(* Logix 5000 project; controller reports 1756-L63 rev 20.11; software revision 20.04; part 7 of 52 *)

        [627].log_data[17].valid := 1, [627].log_data[18].valid := 1, [627].log_data[19].valid := 1, [627].time.Year := 2023, [627].time.Month := 1, [627].time.Day := 14, [627].time.Hour := 5, [627].time.Minute := 14, [627].time.Second := 59, [628].log_data[0].min := 1.0, [628].log_data[0].max := 1.0, [628].log_data[0].total := 900.0, [628].log_data[0].time := 900.0, [628].log_data[0].minminute := 15, [628].log_data[0].maxminute := 15, [628].log_data[0].valid := 1, [628].log_data[1].valid := 1, [628].log_data[2].valid := 1, [628].log_data[3].valid := 1, [628].log_data[4].valid := 1, [628].log_data[5].valid := 1, [628].log_data[6].valid := 1, [628].log_data[7].valid := 1, [628].log_data[8].valid := 1, [628].log_data[9].valid := 1, [628].log_data[10].valid := 1, [628].log_data[11].valid := 1, [628].log_data[12].valid := 1, [628].log_data[13].valid := 1, [628].log_data[14].valid := 1, [628].log_data[15].valid := 1, [628].log_data[16].valid := 1, [628].log_data[17].valid := 1, [628].log_data[18].valid := 1, [628].log_data[19].valid := 1, [628].time.Year := 2023, [628].time.Month := 1, [628].time.Day := 14, [628].time.Hour := 5, [628].time.Minute := 29, [628].time.Second := 59, [629].log_data[0].min := 1.0, [629].log_data[0].max := 1.0, [629].log_data[0].total := 900.0, [629].log_data[0].time := 900.0, [629].log_data[0].minminute := 30, [629].log_data[0].maxminute := 30, [629].log_data[0].valid := 1, [629].log_data[1].valid := 1, [629].log_data[2].valid := 1, [629].log_data[3].valid := 1, [629].log_data[4].valid := 1, [629].log_data[5].valid := 1, [629].log_data[6].valid := 1, [629].log_data[7].valid := 1, [629].log_data[8].valid := 1, [629].log_data[9].valid := 1, [629].log_data[10].valid := 1, [629].log_data[11].valid := 1, [629].log_data[12].valid := 1,
        [629].log_data[13].valid := 1, [629].log_data[14].valid := 1, [629].log_data[15].valid := 1, [629].log_data[16].valid := 1, [629].log_data[17].valid := 1, [629].log_data[18].valid := 1, [629].log_data[19].valid := 1, [629].time.Year := 2023, [629].time.Month := 1, [629].time.Day := 14, [629].time.Hour := 5, [629].time.Minute := 44, [629].time.Second := 59, [630].log_data[0].min := 1.0, [630].log_data[0].max := 1.0, [630].log_data[0].total := 900.0, [630].log_data[0].time := 900.0, [630].log_data[0].minminute := 45, [630].log_data[0].maxminute := 45, [630].log_data[0].valid := 1, [630].log_data[1].valid := 1, [630].log_data[2].valid := 1, [630].log_data[3].valid := 1, [630].log_data[4].valid := 1, [630].log_data[5].valid := 1, [630].log_data[6].valid := 1, [630].log_data[7].valid := 1, [630].log_data[8].valid := 1, [630].log_data[9].valid := 1, [630].log_data[10].valid := 1, [630].log_data[11].valid := 1, [630].log_data[12].valid := 1, [630].log_data[13].valid := 1, [630].log_data[14].valid := 1, [630].log_data[15].valid := 1, [630].log_data[16].valid := 1, [630].log_data[17].valid := 1, [630].log_data[18].valid := 1, [630].log_data[19].valid := 1, [630].time.Year := 2023, [630].time.Month := 1, [630].time.Day := 14, [630].time.Hour := 5, [630].time.Minute := 59, [630].time.Second := 59, [631].log_data[0].min := 1.0, [631].log_data[0].max := 1.0, [631].log_data[0].total := 900.0, [631].log_data[0].time := 900.0, [631].log_data[0].valid := 1, [631].log_data[1].valid := 1, [631].log_data[2].valid := 1, [631].log_data[3].valid := 1, [631].log_data[4].valid := 1, [631].log_data[5].valid := 1, [631].log_data[6].valid := 1, [631].log_data[7].valid := 1, [631].log_data[8].valid := 1, [631].log_data[9].valid := 1, [631].log_data[10].valid := 1,
        [631].log_data[11].valid := 1, [631].log_data[12].valid := 1, [631].log_data[13].valid := 1, [631].log_data[14].valid := 1, [631].log_data[15].valid := 1, [631].log_data[16].valid := 1, [631].log_data[17].valid := 1, [631].log_data[18].valid := 1, [631].log_data[19].valid := 1, [631].time.Year := 2023, [631].time.Month := 1, [631].time.Day := 14, [631].time.Hour := 6, [631].time.Minute := 14, [631].time.Second := 59, [632].log_data[0].min := 1.0, [632].log_data[0].max := 1.0, [632].log_data[0].total := 900.0, [632].log_data[0].time := 900.0, [632].log_data[0].minminute := 15, [632].log_data[0].maxminute := 15, [632].log_data[0].valid := 1, [632].log_data[1].valid := 1, [632].log_data[2].valid := 1, [632].log_data[3].valid := 1, [632].log_data[4].valid := 1, [632].log_data[5].valid := 1, [632].log_data[6].valid := 1, [632].log_data[7].valid := 1, [632].log_data[8].valid := 1, [632].log_data[9].valid := 1, [632].log_data[10].valid := 1, [632].log_data[11].valid := 1, [632].log_data[12].valid := 1, [632].log_data[13].valid := 1, [632].log_data[14].valid := 1, [632].log_data[15].valid := 1, [632].log_data[16].valid := 1, [632].log_data[17].valid := 1, [632].log_data[18].valid := 1, [632].log_data[19].valid := 1, [632].time.Year := 2023, [632].time.Month := 1, [632].time.Day := 14, [632].time.Hour := 6, [632].time.Minute := 29, [632].time.Second := 59, [633].log_data[0].min := 1.0, [633].log_data[0].max := 1.0, [633].log_data[0].total := 900.0, [633].log_data[0].time := 900.0, [633].log_data[0].minminute := 30, [633].log_data[0].maxminute := 30, [633].log_data[0].valid := 1, [633].log_data[1].valid := 1, [633].log_data[2].valid := 1, [633].log_data[3].valid := 1, [633].log_data[4].valid := 1, [633].log_data[5].valid := 1, [633].log_data[6].valid := 1,
        [633].log_data[7].valid := 1, [633].log_data[8].valid := 1, [633].log_data[9].valid := 1, [633].log_data[10].valid := 1, [633].log_data[11].valid := 1, [633].log_data[12].valid := 1, [633].log_data[13].valid := 1, [633].log_data[14].valid := 1, [633].log_data[15].valid := 1, [633].log_data[16].valid := 1, [633].log_data[17].valid := 1, [633].log_data[18].valid := 1, [633].log_data[19].valid := 1, [633].time.Year := 2023, [633].time.Month := 1, [633].time.Day := 14, [633].time.Hour := 6, [633].time.Minute := 44, [633].time.Second := 59, [634].log_data[0].min := 1.0, [634].log_data[0].max := 1.0, [634].log_data[0].total := 900.0, [634].log_data[0].time := 900.0, [634].log_data[0].minminute := 45, [634].log_data[0].maxminute := 45, [634].log_data[0].valid := 1, [634].log_data[1].valid := 1, [634].log_data[2].valid := 1, [634].log_data[3].valid := 1, [634].log_data[4].valid := 1, [634].log_data[5].valid := 1, [634].log_data[6].valid := 1, [634].log_data[7].valid := 1, [634].log_data[8].valid := 1, [634].log_data[9].valid := 1, [634].log_data[10].valid := 1, [634].log_data[11].valid := 1, [634].log_data[12].valid := 1, [634].log_data[13].valid := 1, [634].log_data[14].valid := 1, [634].log_data[15].valid := 1, [634].log_data[16].valid := 1, [634].log_data[17].valid := 1, [634].log_data[18].valid := 1, [634].log_data[19].valid := 1, [634].time.Year := 2023, [634].time.Month := 1, [634].time.Day := 14, [634].time.Hour := 6, [634].time.Minute := 59, [634].time.Second := 59, [635].log_data[0].min := 1.0, [635].log_data[0].max := 1.0, [635].log_data[0].total := 900.0, [635].log_data[0].time := 900.0, [635].log_data[0].valid := 1, [635].log_data[1].valid := 1, [635].log_data[2].valid := 1, [635].log_data[3].valid := 1, [635].log_data[4].valid := 1,
        [635].log_data[5].valid := 1, [635].log_data[6].valid := 1, [635].log_data[7].valid := 1, [635].log_data[8].valid := 1, [635].log_data[9].valid := 1, [635].log_data[10].valid := 1, [635].log_data[11].valid := 1, [635].log_data[12].valid := 1, [635].log_data[13].valid := 1, [635].log_data[14].valid := 1, [635].log_data[15].valid := 1, [635].log_data[16].valid := 1, [635].log_data[17].valid := 1, [635].log_data[18].valid := 1, [635].log_data[19].valid := 1, [635].time.Year := 2023, [635].time.Month := 1, [635].time.Day := 14, [635].time.Hour := 7, [635].time.Minute := 14, [635].time.Second := 59, [636].log_data[0].min := 1.0, [636].log_data[0].max := 1.0, [636].log_data[0].total := 900.0, [636].log_data[0].time := 900.0, [636].log_data[0].minminute := 15, [636].log_data[0].maxminute := 15, [636].log_data[0].valid := 1, [636].log_data[1].valid := 1, [636].log_data[2].valid := 1, [636].log_data[3].valid := 1, [636].log_data[4].valid := 1, [636].log_data[5].valid := 1, [636].log_data[6].valid := 1, [636].log_data[7].valid := 1, [636].log_data[8].valid := 1, [636].log_data[9].valid := 1, [636].log_data[10].valid := 1, [636].log_data[11].valid := 1, [636].log_data[12].valid := 1, [636].log_data[13].valid := 1, [636].log_data[14].valid := 1, [636].log_data[15].valid := 1, [636].log_data[16].valid := 1, [636].log_data[17].valid := 1, [636].log_data[18].valid := 1, [636].log_data[19].valid := 1, [636].time.Year := 2023, [636].time.Month := 1, [636].time.Day := 14, [636].time.Hour := 7, [636].time.Minute := 29, [636].time.Second := 59, [637].log_data[0].min := 1.0, [637].log_data[0].max := 1.0, [637].log_data[0].total := 900.0, [637].log_data[0].time := 900.0, [637].log_data[0].minminute := 30, [637].log_data[0].maxminute := 30, [637].log_data[0].valid := 1,
        [637].log_data[1].valid := 1, [637].log_data[2].valid := 1, [637].log_data[3].valid := 1, [637].log_data[4].valid := 1, [637].log_data[5].valid := 1, [637].log_data[6].valid := 1, [637].log_data[7].valid := 1, [637].log_data[8].valid := 1, [637].log_data[9].valid := 1, [637].log_data[10].valid := 1, [637].log_data[11].valid := 1, [637].log_data[12].valid := 1, [637].log_data[13].valid := 1, [637].log_data[14].valid := 1, [637].log_data[15].valid := 1, [637].log_data[16].valid := 1, [637].log_data[17].valid := 1, [637].log_data[18].valid := 1, [637].log_data[19].valid := 1, [637].time.Year := 2023, [637].time.Month := 1, [637].time.Day := 14, [637].time.Hour := 7, [637].time.Minute := 44, [637].time.Second := 59, [638].log_data[0].min := 1.0, [638].log_data[0].max := 1.0, [638].log_data[0].total := 900.0, [638].log_data[0].time := 900.0, [638].log_data[0].minminute := 45, [638].log_data[0].maxminute := 45, [638].log_data[0].valid := 1, [638].log_data[1].valid := 1, [638].log_data[2].valid := 1, [638].log_data[3].valid := 1, [638].log_data[4].valid := 1, [638].log_data[5].valid := 1, [638].log_data[6].valid := 1, [638].log_data[7].valid := 1, [638].log_data[8].valid := 1, [638].log_data[9].valid := 1, [638].log_data[10].valid := 1, [638].log_data[11].valid := 1, [638].log_data[12].valid := 1, [638].log_data[13].valid := 1, [638].log_data[14].valid := 1, [638].log_data[15].valid := 1, [638].log_data[16].valid := 1, [638].log_data[17].valid := 1, [638].log_data[18].valid := 1, [638].log_data[19].valid := 1, [638].time.Year := 2023, [638].time.Month := 1, [638].time.Day := 14, [638].time.Hour := 7, [638].time.Minute := 59, [638].time.Second := 59, [639].log_data[0].min := 1.0, [639].log_data[0].max := 1.0, [639].log_data[0].total := 900.0,
        [639].log_data[0].time := 900.0, [639].log_data[0].valid := 1, [639].log_data[1].valid := 1, [639].log_data[2].valid := 1, [639].log_data[3].valid := 1, [639].log_data[4].valid := 1, [639].log_data[5].valid := 1, [639].log_data[6].valid := 1, [639].log_data[7].valid := 1, [639].log_data[8].valid := 1, [639].log_data[9].valid := 1, [639].log_data[10].valid := 1, [639].log_data[11].valid := 1, [639].log_data[12].valid := 1, [639].log_data[13].valid := 1, [639].log_data[14].valid := 1, [639].log_data[15].valid := 1, [639].log_data[16].valid := 1, [639].log_data[17].valid := 1, [639].log_data[18].valid := 1, [639].log_data[19].valid := 1, [639].time.Year := 2023, [639].time.Month := 1, [639].time.Day := 14, [639].time.Hour := 8, [639].time.Minute := 14, [639].time.Second := 59, [640].log_data[0].min := 1.0, [640].log_data[0].max := 1.0, [640].log_data[0].total := 900.0, [640].log_data[0].time := 900.0, [640].log_data[0].minminute := 15, [640].log_data[0].maxminute := 15, [640].log_data[0].valid := 1, [640].log_data[1].valid := 1, [640].log_data[2].valid := 1, [640].log_data[3].valid := 1, [640].log_data[4].valid := 1, [640].log_data[5].valid := 1, [640].log_data[6].valid := 1, [640].log_data[7].valid := 1, [640].log_data[8].valid := 1, [640].log_data[9].valid := 1, [640].log_data[10].valid := 1, [640].log_data[11].valid := 1, [640].log_data[12].valid := 1, [640].log_data[13].valid := 1, [640].log_data[14].valid := 1, [640].log_data[15].valid := 1, [640].log_data[16].valid := 1, [640].log_data[17].valid := 1, [640].log_data[18].valid := 1, [640].log_data[19].valid := 1, [640].time.Year := 2023, [640].time.Month := 1, [640].time.Day := 14, [640].time.Hour := 8, [640].time.Minute := 29, [640].time.Second := 59, [641].log_data[0].min := 1.0,
        [641].log_data[0].max := 1.0, [641].log_data[0].total := 900.0, [641].log_data[0].time := 900.0, [641].log_data[0].minminute := 30, [641].log_data[0].maxminute := 30, [641].log_data[0].valid := 1, [641].log_data[1].valid := 1, [641].log_data[2].valid := 1, [641].log_data[3].valid := 1, [641].log_data[4].valid := 1, [641].log_data[5].valid := 1, [641].log_data[6].valid := 1, [641].log_data[7].valid := 1, [641].log_data[8].valid := 1, [641].log_data[9].valid := 1, [641].log_data[10].valid := 1, [641].log_data[11].valid := 1, [641].log_data[12].valid := 1, [641].log_data[13].valid := 1, [641].log_data[14].valid := 1, [641].log_data[15].valid := 1, [641].log_data[16].valid := 1, [641].log_data[17].valid := 1, [641].log_data[18].valid := 1, [641].log_data[19].valid := 1, [641].time.Year := 2023, [641].time.Month := 1, [641].time.Day := 14, [641].time.Hour := 8, [641].time.Minute := 44, [641].time.Second := 59, [642].log_data[0].min := 1.0, [642].log_data[0].max := 1.0, [642].log_data[0].total := 900.0, [642].log_data[0].time := 900.0, [642].log_data[0].minminute := 45, [642].log_data[0].maxminute := 45, [642].log_data[0].valid := 1, [642].log_data[1].valid := 1, [642].log_data[2].valid := 1, [642].log_data[3].valid := 1, [642].log_data[4].valid := 1, [642].log_data[5].valid := 1, [642].log_data[6].valid := 1, [642].log_data[7].valid := 1, [642].log_data[8].valid := 1, [642].log_data[9].valid := 1, [642].log_data[10].valid := 1, [642].log_data[11].valid := 1, [642].log_data[12].valid := 1, [642].log_data[13].valid := 1, [642].log_data[14].valid := 1, [642].log_data[15].valid := 1, [642].log_data[16].valid := 1, [642].log_data[17].valid := 1, [642].log_data[18].valid := 1, [642].log_data[19].valid := 1, [642].time.Year := 2023, [642].time.Month := 1, [642].time.Day := 14,
        [642].time.Hour := 8, [642].time.Minute := 59, [642].time.Second := 59, [643].log_data[0].min := 1.0, [643].log_data[0].max := 1.0, [643].log_data[0].total := 900.0, [643].log_data[0].time := 900.0, [643].log_data[0].valid := 1, [643].log_data[1].valid := 1, [643].log_data[2].valid := 1, [643].log_data[3].valid := 1, [643].log_data[4].valid := 1, [643].log_data[5].valid := 1, [643].log_data[6].valid := 1, [643].log_data[7].valid := 1, [643].log_data[8].valid := 1, [643].log_data[9].valid := 1, [643].log_data[10].valid := 1, [643].log_data[11].valid := 1, [643].log_data[12].valid := 1, [643].log_data[13].valid := 1, [643].log_data[14].valid := 1, [643].log_data[15].valid := 1, [643].log_data[16].valid := 1, [643].log_data[17].valid := 1, [643].log_data[18].valid := 1, [643].log_data[19].valid := 1, [643].time.Year := 2023, [643].time.Month := 1, [643].time.Day := 14, [643].time.Hour := 9, [643].time.Minute := 14, [643].time.Second := 59, [644].log_data[0].min := 1.0, [644].log_data[0].max := 1.0, [644].log_data[0].total := 900.0, [644].log_data[0].time := 900.0, [644].log_data[0].minminute := 15, [644].log_data[0].maxminute := 15, [644].log_data[0].valid := 1, [644].log_data[1].valid := 1, [644].log_data[2].valid := 1, [644].log_data[3].valid := 1, [644].log_data[4].valid := 1, [644].log_data[5].valid := 1, [644].log_data[6].valid := 1, [644].log_data[7].valid := 1, [644].log_data[8].valid := 1, [644].log_data[9].valid := 1, [644].log_data[10].valid := 1, [644].log_data[11].valid := 1, [644].log_data[12].valid := 1, [644].log_data[13].valid := 1, [644].log_data[14].valid := 1, [644].log_data[15].valid := 1, [644].log_data[16].valid := 1, [644].log_data[17].valid := 1, [644].log_data[18].valid := 1, [644].log_data[19].valid := 1, [644].time.Year := 2023,
        [644].time.Month := 1, [644].time.Day := 14, [644].time.Hour := 9, [644].time.Minute := 29, [644].time.Second := 59, [645].log_data[0].min := 1.0, [645].log_data[0].max := 1.0, [645].log_data[0].total := 900.0, [645].log_data[0].time := 900.0, [645].log_data[0].minminute := 30, [645].log_data[0].maxminute := 30, [645].log_data[0].valid := 1, [645].log_data[1].valid := 1, [645].log_data[2].valid := 1, [645].log_data[3].valid := 1, [645].log_data[4].valid := 1, [645].log_data[5].valid := 1, [645].log_data[6].valid := 1, [645].log_data[7].valid := 1, [645].log_data[8].valid := 1, [645].log_data[9].valid := 1, [645].log_data[10].valid := 1, [645].log_data[11].valid := 1, [645].log_data[12].valid := 1, [645].log_data[13].valid := 1, [645].log_data[14].valid := 1, [645].log_data[15].valid := 1, [645].log_data[16].valid := 1, [645].log_data[17].valid := 1, [645].log_data[18].valid := 1, [645].log_data[19].valid := 1, [645].time.Year := 2023, [645].time.Month := 1, [645].time.Day := 14, [645].time.Hour := 9, [645].time.Minute := 44, [645].time.Second := 59, [646].log_data[0].min := 1.0, [646].log_data[0].max := 1.0, [646].log_data[0].total := 900.0, [646].log_data[0].time := 900.0, [646].log_data[0].minminute := 45, [646].log_data[0].maxminute := 45, [646].log_data[0].valid := 1, [646].log_data[1].valid := 1, [646].log_data[2].valid := 1, [646].log_data[3].valid := 1, [646].log_data[4].valid := 1, [646].log_data[5].valid := 1, [646].log_data[6].valid := 1, [646].log_data[7].valid := 1, [646].log_data[8].valid := 1, [646].log_data[9].valid := 1, [646].log_data[10].valid := 1, [646].log_data[11].valid := 1, [646].log_data[12].valid := 1, [646].log_data[13].valid := 1, [646].log_data[14].valid := 1, [646].log_data[15].valid := 1, [646].log_data[16].valid := 1,
        [646].log_data[17].valid := 1, [646].log_data[18].valid := 1, [646].log_data[19].valid := 1, [646].time.Year := 2023, [646].time.Month := 1, [646].time.Day := 14, [646].time.Hour := 9, [646].time.Minute := 59, [646].time.Second := 59, [647].log_data[0].min := 1.0, [647].log_data[0].max := 1.0, [647].log_data[0].total := 900.0, [647].log_data[0].time := 900.0, [647].log_data[0].valid := 1, [647].log_data[1].valid := 1, [647].log_data[2].valid := 1, [647].log_data[3].valid := 1, [647].log_data[4].valid := 1, [647].log_data[5].valid := 1, [647].log_data[6].valid := 1, [647].log_data[7].valid := 1, [647].log_data[8].valid := 1, [647].log_data[9].valid := 1, [647].log_data[10].valid := 1, [647].log_data[11].valid := 1, [647].log_data[12].valid := 1, [647].log_data[13].valid := 1, [647].log_data[14].valid := 1, [647].log_data[15].valid := 1, [647].log_data[16].valid := 1, [647].log_data[17].valid := 1, [647].log_data[18].valid := 1, [647].log_data[19].valid := 1, [647].time.Year := 2023, [647].time.Month := 1, [647].time.Day := 14, [647].time.Hour := 10, [647].time.Minute := 14, [647].time.Second := 59, [648].log_data[0].min := 1.0, [648].log_data[0].max := 1.0, [648].log_data[0].total := 900.0, [648].log_data[0].time := 900.0, [648].log_data[0].minminute := 15, [648].log_data[0].maxminute := 15, [648].log_data[0].valid := 1, [648].log_data[1].valid := 1, [648].log_data[2].valid := 1, [648].log_data[3].valid := 1, [648].log_data[4].valid := 1, [648].log_data[5].valid := 1, [648].log_data[6].valid := 1, [648].log_data[7].valid := 1, [648].log_data[8].valid := 1, [648].log_data[9].valid := 1, [648].log_data[10].valid := 1, [648].log_data[11].valid := 1, [648].log_data[12].valid := 1, [648].log_data[13].valid := 1, [648].log_data[14].valid := 1,
        [648].log_data[15].valid := 1, [648].log_data[16].valid := 1, [648].log_data[17].valid := 1, [648].log_data[18].valid := 1, [648].log_data[19].valid := 1, [648].time.Year := 2023, [648].time.Month := 1, [648].time.Day := 14, [648].time.Hour := 10, [648].time.Minute := 29, [648].time.Second := 59, [649].log_data[0].min := 1.0, [649].log_data[0].max := 1.0, [649].log_data[0].total := 900.0, [649].log_data[0].time := 900.0, [649].log_data[0].minminute := 30, [649].log_data[0].maxminute := 30, [649].log_data[0].valid := 1, [649].log_data[1].valid := 1, [649].log_data[2].valid := 1, [649].log_data[3].valid := 1, [649].log_data[4].valid := 1, [649].log_data[5].valid := 1, [649].log_data[6].valid := 1, [649].log_data[7].valid := 1, [649].log_data[8].valid := 1, [649].log_data[9].valid := 1, [649].log_data[10].valid := 1, [649].log_data[11].valid := 1, [649].log_data[12].valid := 1, [649].log_data[13].valid := 1, [649].log_data[14].valid := 1, [649].log_data[15].valid := 1, [649].log_data[16].valid := 1, [649].log_data[17].valid := 1, [649].log_data[18].valid := 1, [649].log_data[19].valid := 1, [649].time.Year := 2023, [649].time.Month := 1, [649].time.Day := 14, [649].time.Hour := 10, [649].time.Minute := 44, [649].time.Second := 59, [650].log_data[0].min := 1.0, [650].log_data[0].max := 1.0, [650].log_data[0].total := 900.0, [650].log_data[0].time := 900.0, [650].log_data[0].minminute := 45, [650].log_data[0].maxminute := 45, [650].log_data[0].valid := 1, [650].log_data[1].valid := 1, [650].log_data[2].valid := 1, [650].log_data[3].valid := 1, [650].log_data[4].valid := 1, [650].log_data[5].valid := 1, [650].log_data[6].valid := 1, [650].log_data[7].valid := 1, [650].log_data[8].valid := 1, [650].log_data[9].valid := 1, [650].log_data[10].valid := 1,
        [650].log_data[11].valid := 1, [650].log_data[12].valid := 1, [650].log_data[13].valid := 1, [650].log_data[14].valid := 1, [650].log_data[15].valid := 1, [650].log_data[16].valid := 1, [650].log_data[17].valid := 1, [650].log_data[18].valid := 1, [650].log_data[19].valid := 1, [650].time.Year := 2023, [650].time.Month := 1, [650].time.Day := 14, [650].time.Hour := 10, [650].time.Minute := 59, [650].time.Second := 59, [651].log_data[0].min := 1.0, [651].log_data[0].max := 1.0, [651].log_data[0].total := 900.0, [651].log_data[0].time := 900.0, [651].log_data[0].valid := 1, [651].log_data[1].valid := 1, [651].log_data[2].valid := 1, [651].log_data[3].valid := 1, [651].log_data[4].valid := 1, [651].log_data[5].valid := 1, [651].log_data[6].valid := 1, [651].log_data[7].valid := 1, [651].log_data[8].valid := 1, [651].log_data[9].valid := 1, [651].log_data[10].valid := 1, [651].log_data[11].valid := 1, [651].log_data[12].valid := 1, [651].log_data[13].valid := 1, [651].log_data[14].valid := 1, [651].log_data[15].valid := 1, [651].log_data[16].valid := 1, [651].log_data[17].valid := 1, [651].log_data[18].valid := 1, [651].log_data[19].valid := 1, [651].time.Year := 2023, [651].time.Month := 1, [651].time.Day := 14, [651].time.Hour := 11, [651].time.Minute := 14, [651].time.Second := 59, [652].log_data[0].min := 1.0, [652].log_data[0].max := 1.0, [652].log_data[0].total := 900.0, [652].log_data[0].time := 900.0, [652].log_data[0].minminute := 15, [652].log_data[0].maxminute := 15, [652].log_data[0].valid := 1, [652].log_data[1].valid := 1, [652].log_data[2].valid := 1, [652].log_data[3].valid := 1, [652].log_data[4].valid := 1, [652].log_data[5].valid := 1, [652].log_data[6].valid := 1, [652].log_data[7].valid := 1, [652].log_data[8].valid := 1,
        [652].log_data[9].valid := 1, [652].log_data[10].valid := 1, [652].log_data[11].valid := 1, [652].log_data[12].valid := 1, [652].log_data[13].valid := 1, [652].log_data[14].valid := 1, [652].log_data[15].valid := 1, [652].log_data[16].valid := 1, [652].log_data[17].valid := 1, [652].log_data[18].valid := 1, [652].log_data[19].valid := 1, [652].time.Year := 2023, [652].time.Month := 1, [652].time.Day := 14, [652].time.Hour := 11, [652].time.Minute := 29, [652].time.Second := 59, [653].log_data[0].min := 1.0, [653].log_data[0].max := 1.0, [653].log_data[0].total := 900.0, [653].log_data[0].time := 900.0, [653].log_data[0].minminute := 30, [653].log_data[0].maxminute := 30, [653].log_data[0].valid := 1, [653].log_data[1].valid := 1, [653].log_data[2].valid := 1, [653].log_data[3].valid := 1, [653].log_data[4].valid := 1, [653].log_data[5].valid := 1, [653].log_data[6].valid := 1, [653].log_data[7].valid := 1, [653].log_data[8].valid := 1, [653].log_data[9].valid := 1, [653].log_data[10].valid := 1, [653].log_data[11].valid := 1, [653].log_data[12].valid := 1, [653].log_data[13].valid := 1, [653].log_data[14].valid := 1, [653].log_data[15].valid := 1, [653].log_data[16].valid := 1, [653].log_data[17].valid := 1, [653].log_data[18].valid := 1, [653].log_data[19].valid := 1, [653].time.Year := 2023, [653].time.Month := 1, [653].time.Day := 14, [653].time.Hour := 11, [653].time.Minute := 44, [653].time.Second := 59, [654].log_data[0].min := 1.0, [654].log_data[0].max := 1.0, [654].log_data[0].total := 900.0, [654].log_data[0].time := 900.0, [654].log_data[0].minminute := 45, [654].log_data[0].maxminute := 45, [654].log_data[0].valid := 1, [654].log_data[1].valid := 1, [654].log_data[2].valid := 1, [654].log_data[3].valid := 1, [654].log_data[4].valid := 1,
        [654].log_data[5].valid := 1, [654].log_data[6].valid := 1, [654].log_data[7].valid := 1, [654].log_data[8].valid := 1, [654].log_data[9].valid := 1, [654].log_data[10].valid := 1, [654].log_data[11].valid := 1, [654].log_data[12].valid := 1, [654].log_data[13].valid := 1, [654].log_data[14].valid := 1, [654].log_data[15].valid := 1, [654].log_data[16].valid := 1, [654].log_data[17].valid := 1, [654].log_data[18].valid := 1, [654].log_data[19].valid := 1, [654].time.Year := 2023, [654].time.Month := 1, [654].time.Day := 14, [654].time.Hour := 11, [654].time.Minute := 59, [654].time.Second := 59, [655].log_data[0].min := 1.0, [655].log_data[0].max := 1.0, [655].log_data[0].total := 899.5, [655].log_data[0].time := 899.5, [655].log_data[0].valid := 1, [655].log_data[1].valid := 1, [655].log_data[2].valid := 1, [655].log_data[3].valid := 1, [655].log_data[4].valid := 1, [655].log_data[5].valid := 1, [655].log_data[6].valid := 1, [655].log_data[7].valid := 1, [655].log_data[8].valid := 1, [655].log_data[9].valid := 1, [655].log_data[10].valid := 1, [655].log_data[11].valid := 1, [655].log_data[12].valid := 1, [655].log_data[13].valid := 1, [655].log_data[14].valid := 1, [655].log_data[15].valid := 1, [655].log_data[16].valid := 1, [655].log_data[17].valid := 1, [655].log_data[18].valid := 1, [655].log_data[19].valid := 1, [655].time.Year := 2023, [655].time.Month := 1, [655].time.Day := 14, [655].time.Hour := 12, [655].time.Minute := 14, [655].time.Second := 59, [656].log_data[0].min := 1.0, [656].log_data[0].max := 1.0, [656].log_data[0].total := 900.0, [656].log_data[0].time := 900.0, [656].log_data[0].minminute := 15, [656].log_data[0].maxminute := 15, [656].log_data[0].valid := 1, [656].log_data[1].valid := 1, [656].log_data[2].valid := 1,
        [656].log_data[3].valid := 1, [656].log_data[4].valid := 1, [656].log_data[5].valid := 1, [656].log_data[6].valid := 1, [656].log_data[7].valid := 1, [656].log_data[8].valid := 1, [656].log_data[9].valid := 1, [656].log_data[10].valid := 1, [656].log_data[11].valid := 1, [656].log_data[12].valid := 1, [656].log_data[13].valid := 1, [656].log_data[14].valid := 1, [656].log_data[15].valid := 1, [656].log_data[16].valid := 1, [656].log_data[17].valid := 1, [656].log_data[18].valid := 1, [656].log_data[19].valid := 1, [656].time.Year := 2023, [656].time.Month := 1, [656].time.Day := 14, [656].time.Hour := 12, [656].time.Minute := 29, [656].time.Second := 59, [657].log_data[0].min := 1.0, [657].log_data[0].max := 1.0, [657].log_data[0].total := 900.0, [657].log_data[0].time := 900.0, [657].log_data[0].minminute := 30, [657].log_data[0].maxminute := 30, [657].log_data[0].valid := 1, [657].log_data[1].valid := 1, [657].log_data[2].valid := 1, [657].log_data[3].valid := 1, [657].log_data[4].valid := 1, [657].log_data[5].valid := 1, [657].log_data[6].valid := 1, [657].log_data[7].valid := 1, [657].log_data[8].valid := 1, [657].log_data[9].valid := 1, [657].log_data[10].valid := 1, [657].log_data[11].valid := 1, [657].log_data[12].valid := 1, [657].log_data[13].valid := 1, [657].log_data[14].valid := 1, [657].log_data[15].valid := 1, [657].log_data[16].valid := 1, [657].log_data[17].valid := 1, [657].log_data[18].valid := 1, [657].log_data[19].valid := 1, [657].time.Year := 2023, [657].time.Month := 1, [657].time.Day := 14, [657].time.Hour := 12, [657].time.Minute := 44, [657].time.Second := 59, [658].log_data[0].min := 1.0, [658].log_data[0].max := 1.0, [658].log_data[0].total := 900.0, [658].log_data[0].time := 900.0, [658].log_data[0].minminute := 45,
        [658].log_data[0].maxminute := 45, [658].log_data[0].valid := 1, [658].log_data[1].valid := 1, [658].log_data[2].valid := 1, [658].log_data[3].valid := 1, [658].log_data[4].valid := 1, [658].log_data[5].valid := 1, [658].log_data[6].valid := 1, [658].log_data[7].valid := 1, [658].log_data[8].valid := 1, [658].log_data[9].valid := 1, [658].log_data[10].valid := 1, [658].log_data[11].valid := 1, [658].log_data[12].valid := 1, [658].log_data[13].valid := 1, [658].log_data[14].valid := 1, [658].log_data[15].valid := 1, [658].log_data[16].valid := 1, [658].log_data[17].valid := 1, [658].log_data[18].valid := 1, [658].log_data[19].valid := 1, [658].time.Year := 2023, [658].time.Month := 1, [658].time.Day := 14, [658].time.Hour := 12, [658].time.Minute := 59, [658].time.Second := 59, [659].log_data[0].min := 1.0, [659].log_data[0].max := 1.0, [659].log_data[0].total := 900.0, [659].log_data[0].time := 900.0, [659].log_data[0].valid := 1, [659].log_data[1].valid := 1, [659].log_data[2].valid := 1, [659].log_data[3].valid := 1, [659].log_data[4].valid := 1, [659].log_data[5].valid := 1, [659].log_data[6].valid := 1, [659].log_data[7].valid := 1, [659].log_data[8].valid := 1, [659].log_data[9].valid := 1, [659].log_data[10].valid := 1, [659].log_data[11].valid := 1, [659].log_data[12].valid := 1, [659].log_data[13].valid := 1, [659].log_data[14].valid := 1, [659].log_data[15].valid := 1, [659].log_data[16].valid := 1, [659].log_data[17].valid := 1, [659].log_data[18].valid := 1, [659].log_data[19].valid := 1, [659].time.Year := 2023, [659].time.Month := 1, [659].time.Day := 14, [659].time.Hour := 13, [659].time.Minute := 14, [659].time.Second := 59, [660].log_data[0].min := 1.0, [660].log_data[0].max := 1.0, [660].log_data[0].total := 900.0,
        [660].log_data[0].time := 900.0, [660].log_data[0].minminute := 15, [660].log_data[0].maxminute := 15, [660].log_data[0].valid := 1, [660].log_data[1].valid := 1, [660].log_data[2].valid := 1, [660].log_data[3].valid := 1, [660].log_data[4].valid := 1, [660].log_data[5].valid := 1, [660].log_data[6].valid := 1, [660].log_data[7].valid := 1, [660].log_data[8].valid := 1, [660].log_data[9].valid := 1, [660].log_data[10].valid := 1, [660].log_data[11].valid := 1, [660].log_data[12].valid := 1, [660].log_data[13].valid := 1, [660].log_data[14].valid := 1, [660].log_data[15].valid := 1, [660].log_data[16].valid := 1, [660].log_data[17].valid := 1, [660].log_data[18].valid := 1, [660].log_data[19].valid := 1, [660].time.Year := 2023, [660].time.Month := 1, [660].time.Day := 14, [660].time.Hour := 13, [660].time.Minute := 29, [660].time.Second := 59, [661].log_data[0].min := 1.0, [661].log_data[0].max := 1.0, [661].log_data[0].total := 900.0, [661].log_data[0].time := 900.0, [661].log_data[0].minminute := 30, [661].log_data[0].maxminute := 30, [661].log_data[0].valid := 1, [661].log_data[1].valid := 1, [661].log_data[2].valid := 1, [661].log_data[3].valid := 1, [661].log_data[4].valid := 1, [661].log_data[5].valid := 1, [661].log_data[6].valid := 1, [661].log_data[7].valid := 1, [661].log_data[8].valid := 1, [661].log_data[9].valid := 1, [661].log_data[10].valid := 1, [661].log_data[11].valid := 1, [661].log_data[12].valid := 1, [661].log_data[13].valid := 1, [661].log_data[14].valid := 1, [661].log_data[15].valid := 1, [661].log_data[16].valid := 1, [661].log_data[17].valid := 1, [661].log_data[18].valid := 1, [661].log_data[19].valid := 1, [661].time.Year := 2023, [661].time.Month := 1, [661].time.Day := 14, [661].time.Hour := 13, [661].time.Minute := 44,
        [661].time.Second := 59, [662].log_data[0].min := 1.0, [662].log_data[0].max := 1.0, [662].log_data[0].total := 900.0, [662].log_data[0].time := 900.0, [662].log_data[0].minminute := 45, [662].log_data[0].maxminute := 45, [662].log_data[0].valid := 1, [662].log_data[1].valid := 1, [662].log_data[2].valid := 1, [662].log_data[3].valid := 1, [662].log_data[4].valid := 1, [662].log_data[5].valid := 1, [662].log_data[6].valid := 1, [662].log_data[7].valid := 1, [662].log_data[8].valid := 1, [662].log_data[9].valid := 1, [662].log_data[10].valid := 1, [662].log_data[11].valid := 1, [662].log_data[12].valid := 1, [662].log_data[13].valid := 1, [662].log_data[14].valid := 1, [662].log_data[15].valid := 1, [662].log_data[16].valid := 1, [662].log_data[17].valid := 1, [662].log_data[18].valid := 1, [662].log_data[19].valid := 1, [662].time.Year := 2023, [662].time.Month := 1, [662].time.Day := 14, [662].time.Hour := 13, [662].time.Minute := 59, [662].time.Second := 59, [663].log_data[0].min := 1.0, [663].log_data[0].max := 1.0, [663].log_data[0].total := 900.0, [663].log_data[0].time := 900.0, [663].log_data[0].valid := 1, [663].log_data[1].valid := 1, [663].log_data[2].valid := 1, [663].log_data[3].valid := 1, [663].log_data[4].valid := 1, [663].log_data[5].valid := 1, [663].log_data[6].valid := 1, [663].log_data[7].valid := 1, [663].log_data[8].valid := 1, [663].log_data[9].valid := 1, [663].log_data[10].valid := 1, [663].log_data[11].valid := 1, [663].log_data[12].valid := 1, [663].log_data[13].valid := 1, [663].log_data[14].valid := 1, [663].log_data[15].valid := 1, [663].log_data[16].valid := 1, [663].log_data[17].valid := 1, [663].log_data[18].valid := 1, [663].log_data[19].valid := 1, [663].time.Year := 2023, [663].time.Month := 1, [663].time.Day := 14,
        [663].time.Hour := 14, [663].time.Minute := 14, [663].time.Second := 59, [664].log_data[0].min := 1.0, [664].log_data[0].max := 1.0, [664].log_data[0].total := 900.0, [664].log_data[0].time := 900.0, [664].log_data[0].minminute := 15, [664].log_data[0].maxminute := 15, [664].log_data[0].valid := 1, [664].log_data[1].valid := 1, [664].log_data[2].valid := 1, [664].log_data[3].valid := 1, [664].log_data[4].valid := 1, [664].log_data[5].valid := 1, [664].log_data[6].valid := 1, [664].log_data[7].valid := 1, [664].log_data[8].valid := 1, [664].log_data[9].valid := 1, [664].log_data[10].valid := 1, [664].log_data[11].valid := 1, [664].log_data[12].valid := 1, [664].log_data[13].valid := 1, [664].log_data[14].valid := 1, [664].log_data[15].valid := 1, [664].log_data[16].valid := 1, [664].log_data[17].valid := 1, [664].log_data[18].valid := 1, [664].log_data[19].valid := 1, [664].time.Year := 2023, [664].time.Month := 1, [664].time.Day := 14, [664].time.Hour := 14, [664].time.Minute := 29, [664].time.Second := 59, [665].log_data[0].min := 1.0, [665].log_data[0].max := 1.0, [665].log_data[0].total := 900.0, [665].log_data[0].time := 900.0, [665].log_data[0].minminute := 30, [665].log_data[0].maxminute := 30, [665].log_data[0].valid := 1, [665].log_data[1].valid := 1, [665].log_data[2].valid := 1, [665].log_data[3].valid := 1, [665].log_data[4].valid := 1, [665].log_data[5].valid := 1, [665].log_data[6].valid := 1, [665].log_data[7].valid := 1, [665].log_data[8].valid := 1, [665].log_data[9].valid := 1, [665].log_data[10].valid := 1, [665].log_data[11].valid := 1, [665].log_data[12].valid := 1, [665].log_data[13].valid := 1, [665].log_data[14].valid := 1, [665].log_data[15].valid := 1, [665].log_data[16].valid := 1, [665].log_data[17].valid := 1, [665].log_data[18].valid := 1,
        [665].log_data[19].valid := 1, [665].time.Year := 2023, [665].time.Month := 1, [665].time.Day := 14, [665].time.Hour := 14, [665].time.Minute := 44, [665].time.Second := 59, [666].log_data[0].min := 1.0, [666].log_data[0].max := 1.0, [666].log_data[0].total := 900.0, [666].log_data[0].time := 900.0, [666].log_data[0].minminute := 45, [666].log_data[0].maxminute := 45, [666].log_data[0].valid := 1, [666].log_data[1].valid := 1, [666].log_data[2].valid := 1, [666].log_data[3].valid := 1, [666].log_data[4].valid := 1, [666].log_data[5].valid := 1, [666].log_data[6].valid := 1, [666].log_data[7].valid := 1, [666].log_data[8].valid := 1, [666].log_data[9].valid := 1, [666].log_data[10].valid := 1, [666].log_data[11].valid := 1, [666].log_data[12].valid := 1, [666].log_data[13].valid := 1, [666].log_data[14].valid := 1, [666].log_data[15].valid := 1, [666].log_data[16].valid := 1, [666].log_data[17].valid := 1, [666].log_data[18].valid := 1, [666].log_data[19].valid := 1, [666].time.Year := 2023, [666].time.Month := 1, [666].time.Day := 14, [666].time.Hour := 14, [666].time.Minute := 59, [666].time.Second := 59, [667].log_data[0].min := 1.0, [667].log_data[0].max := 1.0, [667].log_data[0].total := 900.0, [667].log_data[0].time := 900.0, [667].log_data[0].valid := 1, [667].log_data[1].valid := 1, [667].log_data[2].valid := 1, [667].log_data[3].valid := 1, [667].log_data[4].valid := 1, [667].log_data[5].valid := 1, [667].log_data[6].valid := 1, [667].log_data[7].valid := 1, [667].log_data[8].valid := 1, [667].log_data[9].valid := 1, [667].log_data[10].valid := 1, [667].log_data[11].valid := 1, [667].log_data[12].valid := 1, [667].log_data[13].valid := 1, [667].log_data[14].valid := 1, [667].log_data[15].valid := 1, [667].log_data[16].valid := 1,
        [667].log_data[17].valid := 1, [667].log_data[18].valid := 1, [667].log_data[19].valid := 1, [667].time.Year := 2023, [667].time.Month := 1, [667].time.Day := 14, [667].time.Hour := 15, [667].time.Minute := 14, [667].time.Second := 59, [668].log_data[0].min := 1.0, [668].log_data[0].max := 1.0, [668].log_data[0].total := 900.0, [668].log_data[0].time := 900.0, [668].log_data[0].minminute := 15, [668].log_data[0].maxminute := 15, [668].log_data[0].valid := 1, [668].log_data[1].valid := 1, [668].log_data[2].valid := 1, [668].log_data[3].valid := 1, [668].log_data[4].valid := 1, [668].log_data[5].valid := 1, [668].log_data[6].valid := 1, [668].log_data[7].valid := 1, [668].log_data[8].valid := 1, [668].log_data[9].valid := 1, [668].log_data[10].valid := 1, [668].log_data[11].valid := 1, [668].log_data[12].valid := 1, [668].log_data[13].valid := 1, [668].log_data[14].valid := 1, [668].log_data[15].valid := 1, [668].log_data[16].valid := 1, [668].log_data[17].valid := 1, [668].log_data[18].valid := 1, [668].log_data[19].valid := 1, [668].time.Year := 2023, [668].time.Month := 1, [668].time.Day := 14, [668].time.Hour := 15, [668].time.Minute := 29, [668].time.Second := 59, [669].log_data[0].min := 1.0, [669].log_data[0].max := 1.0, [669].log_data[0].total := 900.0, [669].log_data[0].time := 900.0, [669].log_data[0].minminute := 30, [669].log_data[0].maxminute := 30, [669].log_data[0].valid := 1, [669].log_data[1].valid := 1, [669].log_data[2].valid := 1, [669].log_data[3].valid := 1, [669].log_data[4].valid := 1, [669].log_data[5].valid := 1, [669].log_data[6].valid := 1, [669].log_data[7].valid := 1, [669].log_data[8].valid := 1, [669].log_data[9].valid := 1, [669].log_data[10].valid := 1, [669].log_data[11].valid := 1, [669].log_data[12].valid := 1,
        [669].log_data[13].valid := 1, [669].log_data[14].valid := 1, [669].log_data[15].valid := 1, [669].log_data[16].valid := 1, [669].log_data[17].valid := 1, [669].log_data[18].valid := 1, [669].log_data[19].valid := 1, [669].time.Year := 2023, [669].time.Month := 1, [669].time.Day := 14, [669].time.Hour := 15, [669].time.Minute := 44, [669].time.Second := 59, [670].log_data[0].min := 1.0, [670].log_data[0].max := 1.0, [670].log_data[0].total := 900.0, [670].log_data[0].time := 900.0, [670].log_data[0].minminute := 45, [670].log_data[0].maxminute := 45, [670].log_data[0].valid := 1, [670].log_data[1].valid := 1, [670].log_data[2].valid := 1, [670].log_data[3].valid := 1, [670].log_data[4].valid := 1, [670].log_data[5].valid := 1, [670].log_data[6].valid := 1, [670].log_data[7].valid := 1, [670].log_data[8].valid := 1, [670].log_data[9].valid := 1, [670].log_data[10].valid := 1, [670].log_data[11].valid := 1, [670].log_data[12].valid := 1, [670].log_data[13].valid := 1, [670].log_data[14].valid := 1, [670].log_data[15].valid := 1, [670].log_data[16].valid := 1, [670].log_data[17].valid := 1, [670].log_data[18].valid := 1, [670].log_data[19].valid := 1, [670].time.Year := 2023, [670].time.Month := 1, [670].time.Day := 14, [670].time.Hour := 15, [670].time.Minute := 59, [670].time.Second := 59, [671].log_data[0].min := 1.0, [671].log_data[0].max := 1.0, [671].log_data[0].total := 900.0, [671].log_data[0].time := 900.0, [671].log_data[0].valid := 1, [671].log_data[1].valid := 1, [671].log_data[2].valid := 1, [671].log_data[3].valid := 1, [671].log_data[4].valid := 1, [671].log_data[5].valid := 1, [671].log_data[6].valid := 1, [671].log_data[7].valid := 1, [671].log_data[8].valid := 1, [671].log_data[9].valid := 1, [671].log_data[10].valid := 1,
        [671].log_data[11].valid := 1, [671].log_data[12].valid := 1, [671].log_data[13].valid := 1, [671].log_data[14].valid := 1, [671].log_data[15].valid := 1, [671].log_data[16].valid := 1, [671].log_data[17].valid := 1, [671].log_data[18].valid := 1, [671].log_data[19].valid := 1, [671].time.Year := 2023, [671].time.Month := 1, [671].time.Day := 14, [671].time.Hour := 16, [671].time.Minute := 14, [671].time.Second := 59, [672].log_data[0].min := 1.0, [672].log_data[0].max := 1.0, [672].log_data[0].total := 900.0, [672].log_data[0].time := 900.0, [672].log_data[0].minminute := 15, [672].log_data[0].maxminute := 15, [672].log_data[0].valid := 1, [672].log_data[1].valid := 1, [672].log_data[2].valid := 1, [672].log_data[3].valid := 1, [672].log_data[4].valid := 1, [672].log_data[5].valid := 1, [672].log_data[6].valid := 1, [672].log_data[7].valid := 1, [672].log_data[8].valid := 1, [672].log_data[9].valid := 1, [672].log_data[10].valid := 1, [672].log_data[11].valid := 1, [672].log_data[12].valid := 1, [672].log_data[13].valid := 1, [672].log_data[14].valid := 1, [672].log_data[15].valid := 1, [672].log_data[16].valid := 1, [672].log_data[17].valid := 1, [672].log_data[18].valid := 1, [672].log_data[19].valid := 1, [672].time.Year := 2023, [672].time.Month := 1, [672].time.Day := 14, [672].time.Hour := 16, [672].time.Minute := 29, [672].time.Second := 59, [673].log_data[0].min := 1.0, [673].log_data[0].max := 1.0, [673].log_data[0].total := 900.0, [673].log_data[0].time := 900.0, [673].log_data[0].minminute := 30, [673].log_data[0].maxminute := 30, [673].log_data[0].valid := 1, [673].log_data[1].valid := 1, [673].log_data[2].valid := 1, [673].log_data[3].valid := 1, [673].log_data[4].valid := 1, [673].log_data[5].valid := 1, [673].log_data[6].valid := 1,
        [673].log_data[7].valid := 1, [673].log_data[8].valid := 1, [673].log_data[9].valid := 1, [673].log_data[10].valid := 1, [673].log_data[11].valid := 1, [673].log_data[12].valid := 1, [673].log_data[13].valid := 1, [673].log_data[14].valid := 1, [673].log_data[15].valid := 1, [673].log_data[16].valid := 1, [673].log_data[17].valid := 1, [673].log_data[18].valid := 1, [673].log_data[19].valid := 1, [673].time.Year := 2023, [673].time.Month := 1, [673].time.Day := 14, [673].time.Hour := 16, [673].time.Minute := 44, [673].time.Second := 59, [674].log_data[0].min := 1.0, [674].log_data[0].max := 1.0, [674].log_data[0].total := 900.0, [674].log_data[0].time := 900.0, [674].log_data[0].minminute := 45, [674].log_data[0].maxminute := 45, [674].log_data[0].valid := 1, [674].log_data[1].valid := 1, [674].log_data[2].valid := 1, [674].log_data[3].valid := 1, [674].log_data[4].valid := 1, [674].log_data[5].valid := 1, [674].log_data[6].valid := 1, [674].log_data[7].valid := 1, [674].log_data[8].valid := 1, [674].log_data[9].valid := 1, [674].log_data[10].valid := 1, [674].log_data[11].valid := 1, [674].log_data[12].valid := 1, [674].log_data[13].valid := 1, [674].log_data[14].valid := 1, [674].log_data[15].valid := 1, [674].log_data[16].valid := 1, [674].log_data[17].valid := 1, [674].log_data[18].valid := 1, [674].log_data[19].valid := 1, [674].time.Year := 2023, [674].time.Month := 1, [674].time.Day := 14, [674].time.Hour := 16, [674].time.Minute := 59, [674].time.Second := 59, [675].log_data[0].min := 1.0, [675].log_data[0].max := 1.0, [675].log_data[0].total := 900.0, [675].log_data[0].time := 900.0, [675].log_data[0].valid := 1, [675].log_data[1].valid := 1, [675].log_data[2].valid := 1, [675].log_data[3].valid := 1, [675].log_data[4].valid := 1,
        [675].log_data[5].valid := 1, [675].log_data[6].valid := 1, [675].log_data[7].valid := 1, [675].log_data[8].valid := 1, [675].log_data[9].valid := 1, [675].log_data[10].valid := 1, [675].log_data[11].valid := 1, [675].log_data[12].valid := 1, [675].log_data[13].valid := 1, [675].log_data[14].valid := 1, [675].log_data[15].valid := 1, [675].log_data[16].valid := 1, [675].log_data[17].valid := 1, [675].log_data[18].valid := 1, [675].log_data[19].valid := 1, [675].time.Year := 2023, [675].time.Month := 1, [675].time.Day := 14, [675].time.Hour := 17, [675].time.Minute := 14, [675].time.Second := 59, [676].log_data[0].min := 1.0, [676].log_data[0].max := 1.0, [676].log_data[0].total := 900.0, [676].log_data[0].time := 900.0, [676].log_data[0].minminute := 15, [676].log_data[0].maxminute := 15, [676].log_data[0].valid := 1, [676].log_data[1].valid := 1, [676].log_data[2].valid := 1, [676].log_data[3].valid := 1, [676].log_data[4].valid := 1, [676].log_data[5].valid := 1, [676].log_data[6].valid := 1, [676].log_data[7].valid := 1, [676].log_data[8].valid := 1, [676].log_data[9].valid := 1, [676].log_data[10].valid := 1, [676].log_data[11].valid := 1, [676].log_data[12].valid := 1, [676].log_data[13].valid := 1, [676].log_data[14].valid := 1, [676].log_data[15].valid := 1, [676].log_data[16].valid := 1, [676].log_data[17].valid := 1, [676].log_data[18].valid := 1, [676].log_data[19].valid := 1, [676].time.Year := 2023, [676].time.Month := 1, [676].time.Day := 14, [676].time.Hour := 17, [676].time.Minute := 29, [676].time.Second := 59, [677].log_data[0].min := 1.0, [677].log_data[0].max := 1.0, [677].log_data[0].total := 900.0, [677].log_data[0].time := 900.0, [677].log_data[0].minminute := 30, [677].log_data[0].maxminute := 30, [677].log_data[0].valid := 1,
        [677].log_data[1].valid := 1, [677].log_data[2].valid := 1, [677].log_data[3].valid := 1, [677].log_data[4].valid := 1, [677].log_data[5].valid := 1, [677].log_data[6].valid := 1, [677].log_data[7].valid := 1, [677].log_data[8].valid := 1, [677].log_data[9].valid := 1, [677].log_data[10].valid := 1, [677].log_data[11].valid := 1, [677].log_data[12].valid := 1, [677].log_data[13].valid := 1, [677].log_data[14].valid := 1, [677].log_data[15].valid := 1, [677].log_data[16].valid := 1, [677].log_data[17].valid := 1, [677].log_data[18].valid := 1, [677].log_data[19].valid := 1, [677].time.Year := 2023, [677].time.Month := 1, [677].time.Day := 14, [677].time.Hour := 17, [677].time.Minute := 44, [677].time.Second := 59, [678].log_data[0].min := 1.0, [678].log_data[0].max := 1.0, [678].log_data[0].total := 900.0, [678].log_data[0].time := 900.0, [678].log_data[0].minminute := 45, [678].log_data[0].maxminute := 45, [678].log_data[0].valid := 1, [678].log_data[1].valid := 1, [678].log_data[2].valid := 1, [678].log_data[3].valid := 1, [678].log_data[4].valid := 1, [678].log_data[5].valid := 1, [678].log_data[6].valid := 1, [678].log_data[7].valid := 1, [678].log_data[8].valid := 1, [678].log_data[9].valid := 1, [678].log_data[10].valid := 1, [678].log_data[11].valid := 1, [678].log_data[12].valid := 1, [678].log_data[13].valid := 1, [678].log_data[14].valid := 1, [678].log_data[15].valid := 1, [678].log_data[16].valid := 1, [678].log_data[17].valid := 1, [678].log_data[18].valid := 1, [678].log_data[19].valid := 1, [678].time.Year := 2023, [678].time.Month := 1, [678].time.Day := 14, [678].time.Hour := 17, [678].time.Minute := 59, [678].time.Second := 59, [679].log_data[0].min := 1.0, [679].log_data[0].max := 1.0, [679].log_data[0].total := 900.0,
        [679].log_data[0].time := 900.0, [679].log_data[0].valid := 1, [679].log_data[1].valid := 1, [679].log_data[2].valid := 1, [679].log_data[3].valid := 1, [679].log_data[4].valid := 1, [679].log_data[5].valid := 1, [679].log_data[6].valid := 1, [679].log_data[7].valid := 1, [679].log_data[8].valid := 1, [679].log_data[9].valid := 1, [679].log_data[10].valid := 1, [679].log_data[11].valid := 1, [679].log_data[12].valid := 1, [679].log_data[13].valid := 1, [679].log_data[14].valid := 1, [679].log_data[15].valid := 1, [679].log_data[16].valid := 1, [679].log_data[17].valid := 1, [679].log_data[18].valid := 1, [679].log_data[19].valid := 1, [679].time.Year := 2023, [679].time.Month := 1, [679].time.Day := 14, [679].time.Hour := 18, [679].time.Minute := 14, [679].time.Second := 59, [680].log_data[0].min := 1.0, [680].log_data[0].max := 1.0, [680].log_data[0].total := 900.0, [680].log_data[0].time := 900.0, [680].log_data[0].minminute := 15, [680].log_data[0].maxminute := 15, [680].log_data[0].valid := 1, [680].log_data[1].valid := 1, [680].log_data[2].valid := 1, [680].log_data[3].valid := 1, [680].log_data[4].valid := 1, [680].log_data[5].valid := 1, [680].log_data[6].valid := 1, [680].log_data[7].valid := 1, [680].log_data[8].valid := 1, [680].log_data[9].valid := 1, [680].log_data[10].valid := 1, [680].log_data[11].valid := 1, [680].log_data[12].valid := 1, [680].log_data[13].valid := 1, [680].log_data[14].valid := 1, [680].log_data[15].valid := 1, [680].log_data[16].valid := 1, [680].log_data[17].valid := 1, [680].log_data[18].valid := 1, [680].log_data[19].valid := 1, [680].time.Year := 2023, [680].time.Month := 1, [680].time.Day := 14, [680].time.Hour := 18, [680].time.Minute := 29, [680].time.Second := 59, [681].log_data[0].min := 1.0,
        [681].log_data[0].max := 1.0, [681].log_data[0].total := 900.0, [681].log_data[0].time := 900.0, [681].log_data[0].minminute := 30, [681].log_data[0].maxminute := 30, [681].log_data[0].valid := 1, [681].log_data[1].valid := 1, [681].log_data[2].valid := 1, [681].log_data[3].valid := 1, [681].log_data[4].valid := 1, [681].log_data[5].valid := 1, [681].log_data[6].valid := 1, [681].log_data[7].valid := 1, [681].log_data[8].valid := 1, [681].log_data[9].valid := 1, [681].log_data[10].valid := 1, [681].log_data[11].valid := 1, [681].log_data[12].valid := 1, [681].log_data[13].valid := 1, [681].log_data[14].valid := 1, [681].log_data[15].valid := 1, [681].log_data[16].valid := 1, [681].log_data[17].valid := 1, [681].log_data[18].valid := 1, [681].log_data[19].valid := 1, [681].time.Year := 2023, [681].time.Month := 1, [681].time.Day := 14, [681].time.Hour := 18, [681].time.Minute := 44, [681].time.Second := 59, [682].log_data[0].min := 1.0, [682].log_data[0].max := 1.0, [682].log_data[0].total := 900.0, [682].log_data[0].time := 900.0, [682].log_data[0].minminute := 45, [682].log_data[0].maxminute := 45, [682].log_data[0].valid := 1, [682].log_data[1].valid := 1, [682].log_data[2].valid := 1, [682].log_data[3].valid := 1, [682].log_data[4].valid := 1, [682].log_data[5].valid := 1, [682].log_data[6].valid := 1, [682].log_data[7].valid := 1, [682].log_data[8].valid := 1, [682].log_data[9].valid := 1, [682].log_data[10].valid := 1, [682].log_data[11].valid := 1, [682].log_data[12].valid := 1, [682].log_data[13].valid := 1, [682].log_data[14].valid := 1, [682].log_data[15].valid := 1, [682].log_data[16].valid := 1, [682].log_data[17].valid := 1, [682].log_data[18].valid := 1, [682].log_data[19].valid := 1, [682].time.Year := 2023, [682].time.Month := 1, [682].time.Day := 14,
        [682].time.Hour := 18, [682].time.Minute := 59, [682].time.Second := 59, [683].log_data[0].min := 1.0, [683].log_data[0].max := 1.0, [683].log_data[0].total := 900.0, [683].log_data[0].time := 900.0, [683].log_data[0].valid := 1, [683].log_data[1].valid := 1, [683].log_data[2].valid := 1, [683].log_data[3].valid := 1, [683].log_data[4].valid := 1, [683].log_data[5].valid := 1, [683].log_data[6].valid := 1, [683].log_data[7].valid := 1, [683].log_data[8].valid := 1, [683].log_data[9].valid := 1, [683].log_data[10].valid := 1, [683].log_data[11].valid := 1, [683].log_data[12].valid := 1, [683].log_data[13].valid := 1, [683].log_data[14].valid := 1, [683].log_data[15].valid := 1, [683].log_data[16].valid := 1, [683].log_data[17].valid := 1, [683].log_data[18].valid := 1, [683].log_data[19].valid := 1, [683].time.Year := 2023, [683].time.Month := 1, [683].time.Day := 14, [683].time.Hour := 19, [683].time.Minute := 14, [683].time.Second := 59, [684].log_data[0].min := 1.0, [684].log_data[0].max := 1.0, [684].log_data[0].total := 900.0, [684].log_data[0].time := 900.0, [684].log_data[0].minminute := 15, [684].log_data[0].maxminute := 15, [684].log_data[0].valid := 1, [684].log_data[1].valid := 1, [684].log_data[2].valid := 1, [684].log_data[3].valid := 1, [684].log_data[4].valid := 1, [684].log_data[5].valid := 1, [684].log_data[6].valid := 1, [684].log_data[7].valid := 1, [684].log_data[8].valid := 1, [684].log_data[9].valid := 1, [684].log_data[10].valid := 1, [684].log_data[11].valid := 1, [684].log_data[12].valid := 1, [684].log_data[13].valid := 1, [684].log_data[14].valid := 1, [684].log_data[15].valid := 1, [684].log_data[16].valid := 1, [684].log_data[17].valid := 1, [684].log_data[18].valid := 1, [684].log_data[19].valid := 1, [684].time.Year := 2023,
        [684].time.Month := 1, [684].time.Day := 14, [684].time.Hour := 19, [684].time.Minute := 29, [684].time.Second := 59, [685].log_data[0].min := 1.0, [685].log_data[0].max := 1.0, [685].log_data[0].total := 900.0, [685].log_data[0].time := 900.0, [685].log_data[0].minminute := 30, [685].log_data[0].maxminute := 30, [685].log_data[0].valid := 1, [685].log_data[1].valid := 1, [685].log_data[2].valid := 1, [685].log_data[3].valid := 1, [685].log_data[4].valid := 1, [685].log_data[5].valid := 1, [685].log_data[6].valid := 1, [685].log_data[7].valid := 1, [685].log_data[8].valid := 1, [685].log_data[9].valid := 1, [685].log_data[10].valid := 1, [685].log_data[11].valid := 1, [685].log_data[12].valid := 1, [685].log_data[13].valid := 1, [685].log_data[14].valid := 1, [685].log_data[15].valid := 1, [685].log_data[16].valid := 1, [685].log_data[17].valid := 1, [685].log_data[18].valid := 1, [685].log_data[19].valid := 1, [685].time.Year := 2023, [685].time.Month := 1, [685].time.Day := 14, [685].time.Hour := 19, [685].time.Minute := 44, [685].time.Second := 59, [686].log_data[0].min := 1.0, [686].log_data[0].max := 1.0, [686].log_data[0].total := 900.0, [686].log_data[0].time := 900.0, [686].log_data[0].minminute := 45, [686].log_data[0].maxminute := 45, [686].log_data[0].valid := 1, [686].log_data[1].valid := 1, [686].log_data[2].valid := 1, [686].log_data[3].valid := 1, [686].log_data[4].valid := 1, [686].log_data[5].valid := 1, [686].log_data[6].valid := 1, [686].log_data[7].valid := 1, [686].log_data[8].valid := 1, [686].log_data[9].valid := 1, [686].log_data[10].valid := 1, [686].log_data[11].valid := 1, [686].log_data[12].valid := 1, [686].log_data[13].valid := 1, [686].log_data[14].valid := 1, [686].log_data[15].valid := 1, [686].log_data[16].valid := 1,
        [686].log_data[17].valid := 1, [686].log_data[18].valid := 1, [686].log_data[19].valid := 1, [686].time.Year := 2023, [686].time.Month := 1, [686].time.Day := 14, [686].time.Hour := 19, [686].time.Minute := 59, [686].time.Second := 59, [687].log_data[0].min := 1.0, [687].log_data[0].max := 1.0, [687].log_data[0].total := 900.0, [687].log_data[0].time := 900.0, [687].log_data[0].valid := 1, [687].log_data[1].valid := 1, [687].log_data[2].valid := 1, [687].log_data[3].valid := 1, [687].log_data[4].valid := 1, [687].log_data[5].valid := 1, [687].log_data[6].valid := 1, [687].log_data[7].valid := 1, [687].log_data[8].valid := 1, [687].log_data[9].valid := 1, [687].log_data[10].valid := 1, [687].log_data[11].valid := 1, [687].log_data[12].valid := 1, [687].log_data[13].valid := 1, [687].log_data[14].valid := 1, [687].log_data[15].valid := 1, [687].log_data[16].valid := 1, [687].log_data[17].valid := 1, [687].log_data[18].valid := 1, [687].log_data[19].valid := 1, [687].time.Year := 2023, [687].time.Month := 1, [687].time.Day := 14, [687].time.Hour := 20, [687].time.Minute := 14, [687].time.Second := 59, [688].log_data[0].min := 1.0, [688].log_data[0].max := 1.0, [688].log_data[0].total := 900.0, [688].log_data[0].time := 900.0, [688].log_data[0].minminute := 15, [688].log_data[0].maxminute := 15, [688].log_data[0].valid := 1, [688].log_data[1].valid := 1, [688].log_data[2].valid := 1, [688].log_data[3].valid := 1, [688].log_data[4].valid := 1, [688].log_data[5].valid := 1, [688].log_data[6].valid := 1, [688].log_data[7].valid := 1, [688].log_data[8].valid := 1, [688].log_data[9].valid := 1, [688].log_data[10].valid := 1, [688].log_data[11].valid := 1, [688].log_data[12].valid := 1, [688].log_data[13].valid := 1, [688].log_data[14].valid := 1,
        [688].log_data[15].valid := 1, [688].log_data[16].valid := 1, [688].log_data[17].valid := 1, [688].log_data[18].valid := 1, [688].log_data[19].valid := 1, [688].time.Year := 2023, [688].time.Month := 1, [688].time.Day := 14, [688].time.Hour := 20, [688].time.Minute := 29, [688].time.Second := 59, [689].log_data[0].min := 1.0, [689].log_data[0].max := 1.0, [689].log_data[0].total := 900.0, [689].log_data[0].time := 900.0, [689].log_data[0].minminute := 30, [689].log_data[0].maxminute := 30, [689].log_data[0].valid := 1, [689].log_data[1].valid := 1, [689].log_data[2].valid := 1, [689].log_data[3].valid := 1, [689].log_data[4].valid := 1, [689].log_data[5].valid := 1, [689].log_data[6].valid := 1, [689].log_data[7].valid := 1, [689].log_data[8].valid := 1, [689].log_data[9].valid := 1, [689].log_data[10].valid := 1, [689].log_data[11].valid := 1, [689].log_data[12].valid := 1, [689].log_data[13].valid := 1, [689].log_data[14].valid := 1, [689].log_data[15].valid := 1, [689].log_data[16].valid := 1, [689].log_data[17].valid := 1, [689].log_data[18].valid := 1, [689].log_data[19].valid := 1, [689].time.Year := 2023, [689].time.Month := 1, [689].time.Day := 14, [689].time.Hour := 20, [689].time.Minute := 44, [689].time.Second := 59, [690].log_data[0].min := 1.0, [690].log_data[0].max := 1.0, [690].log_data[0].total := 900.0, [690].log_data[0].time := 900.0, [690].log_data[0].minminute := 45, [690].log_data[0].maxminute := 45, [690].log_data[0].valid := 1, [690].log_data[1].valid := 1, [690].log_data[2].valid := 1, [690].log_data[3].valid := 1, [690].log_data[4].valid := 1, [690].log_data[5].valid := 1, [690].log_data[6].valid := 1, [690].log_data[7].valid := 1, [690].log_data[8].valid := 1, [690].log_data[9].valid := 1, [690].log_data[10].valid := 1,
        [690].log_data[11].valid := 1, [690].log_data[12].valid := 1, [690].log_data[13].valid := 1, [690].log_data[14].valid := 1, [690].log_data[15].valid := 1, [690].log_data[16].valid := 1, [690].log_data[17].valid := 1, [690].log_data[18].valid := 1, [690].log_data[19].valid := 1, [690].time.Year := 2023, [690].time.Month := 1, [690].time.Day := 14, [690].time.Hour := 20, [690].time.Minute := 59, [690].time.Second := 59, [691].log_data[0].min := 1.0, [691].log_data[0].max := 1.0, [691].log_data[0].total := 900.0, [691].log_data[0].time := 900.0, [691].log_data[0].valid := 1, [691].log_data[1].valid := 1, [691].log_data[2].valid := 1, [691].log_data[3].valid := 1, [691].log_data[4].valid := 1, [691].log_data[5].valid := 1, [691].log_data[6].valid := 1, [691].log_data[7].valid := 1, [691].log_data[8].valid := 1, [691].log_data[9].valid := 1, [691].log_data[10].valid := 1, [691].log_data[11].valid := 1, [691].log_data[12].valid := 1, [691].log_data[13].valid := 1, [691].log_data[14].valid := 1, [691].log_data[15].valid := 1, [691].log_data[16].valid := 1, [691].log_data[17].valid := 1, [691].log_data[18].valid := 1, [691].log_data[19].valid := 1, [691].time.Year := 2023, [691].time.Month := 1, [691].time.Day := 14, [691].time.Hour := 21, [691].time.Minute := 14, [691].time.Second := 59, [692].log_data[0].min := 1.0, [692].log_data[0].max := 1.0, [692].log_data[0].total := 900.0, [692].log_data[0].time := 900.0, [692].log_data[0].minminute := 15, [692].log_data[0].maxminute := 15, [692].log_data[0].valid := 1, [692].log_data[1].valid := 1, [692].log_data[2].valid := 1, [692].log_data[3].valid := 1, [692].log_data[4].valid := 1, [692].log_data[5].valid := 1, [692].log_data[6].valid := 1, [692].log_data[7].valid := 1, [692].log_data[8].valid := 1,
        [692].log_data[9].valid := 1, [692].log_data[10].valid := 1, [692].log_data[11].valid := 1, [692].log_data[12].valid := 1, [692].log_data[13].valid := 1, [692].log_data[14].valid := 1, [692].log_data[15].valid := 1, [692].log_data[16].valid := 1, [692].log_data[17].valid := 1, [692].log_data[18].valid := 1, [692].log_data[19].valid := 1, [692].time.Year := 2023, [692].time.Month := 1, [692].time.Day := 14, [692].time.Hour := 21, [692].time.Minute := 29, [692].time.Second := 59, [693].log_data[0].min := 1.0, [693].log_data[0].max := 1.0, [693].log_data[0].total := 900.0, [693].log_data[0].time := 900.0, [693].log_data[0].minminute := 30, [693].log_data[0].maxminute := 30, [693].log_data[0].valid := 1, [693].log_data[1].valid := 1, [693].log_data[2].valid := 1, [693].log_data[3].valid := 1, [693].log_data[4].valid := 1, [693].log_data[5].valid := 1, [693].log_data[6].valid := 1, [693].log_data[7].valid := 1, [693].log_data[8].valid := 1, [693].log_data[9].valid := 1, [693].log_data[10].valid := 1, [693].log_data[11].valid := 1, [693].log_data[12].valid := 1, [693].log_data[13].valid := 1, [693].log_data[14].valid := 1, [693].log_data[15].valid := 1, [693].log_data[16].valid := 1, [693].log_data[17].valid := 1, [693].log_data[18].valid := 1, [693].log_data[19].valid := 1, [693].time.Year := 2023, [693].time.Month := 1, [693].time.Day := 14, [693].time.Hour := 21, [693].time.Minute := 44, [693].time.Second := 59, [694].log_data[0].min := 1.0, [694].log_data[0].max := 1.0, [694].log_data[0].total := 900.0, [694].log_data[0].time := 900.0, [694].log_data[0].minminute := 45, [694].log_data[0].maxminute := 45, [694].log_data[0].valid := 1, [694].log_data[1].valid := 1, [694].log_data[2].valid := 1, [694].log_data[3].valid := 1, [694].log_data[4].valid := 1,
        [694].log_data[5].valid := 1, [694].log_data[6].valid := 1, [694].log_data[7].valid := 1, [694].log_data[8].valid := 1, [694].log_data[9].valid := 1, [694].log_data[10].valid := 1, [694].log_data[11].valid := 1, [694].log_data[12].valid := 1, [694].log_data[13].valid := 1, [694].log_data[14].valid := 1, [694].log_data[15].valid := 1, [694].log_data[16].valid := 1, [694].log_data[17].valid := 1, [694].log_data[18].valid := 1, [694].log_data[19].valid := 1, [694].time.Year := 2023, [694].time.Month := 1, [694].time.Day := 14, [694].time.Hour := 21, [694].time.Minute := 59, [694].time.Second := 59, [695].log_data[0].min := 1.0, [695].log_data[0].max := 1.0, [695].log_data[0].total := 900.0, [695].log_data[0].time := 900.0, [695].log_data[0].valid := 1, [695].log_data[1].valid := 1, [695].log_data[2].valid := 1, [695].log_data[3].valid := 1, [695].log_data[4].valid := 1, [695].log_data[5].valid := 1, [695].log_data[6].valid := 1, [695].log_data[7].valid := 1, [695].log_data[8].valid := 1, [695].log_data[9].valid := 1, [695].log_data[10].valid := 1, [695].log_data[11].valid := 1, [695].log_data[12].valid := 1, [695].log_data[13].valid := 1, [695].log_data[14].valid := 1, [695].log_data[15].valid := 1, [695].log_data[16].valid := 1, [695].log_data[17].valid := 1, [695].log_data[18].valid := 1, [695].log_data[19].valid := 1, [695].time.Year := 2023, [695].time.Month := 1, [695].time.Day := 14, [695].time.Hour := 22, [695].time.Minute := 14, [695].time.Second := 59, [696].log_data[0].min := 1.0, [696].log_data[0].max := 1.0, [696].log_data[0].total := 900.0, [696].log_data[0].time := 900.0, [696].log_data[0].minminute := 15, [696].log_data[0].maxminute := 15, [696].log_data[0].valid := 1, [696].log_data[1].valid := 1, [696].log_data[2].valid := 1,
        [696].log_data[3].valid := 1, [696].log_data[4].valid := 1, [696].log_data[5].valid := 1, [696].log_data[6].valid := 1, [696].log_data[7].valid := 1, [696].log_data[8].valid := 1, [696].log_data[9].valid := 1, [696].log_data[10].valid := 1, [696].log_data[11].valid := 1, [696].log_data[12].valid := 1, [696].log_data[13].valid := 1, [696].log_data[14].valid := 1, [696].log_data[15].valid := 1, [696].log_data[16].valid := 1, [696].log_data[17].valid := 1, [696].log_data[18].valid := 1, [696].log_data[19].valid := 1, [696].time.Year := 2023, [696].time.Month := 1, [696].time.Day := 14, [696].time.Hour := 22, [696].time.Minute := 29, [696].time.Second := 59, [697].log_data[0].min := 1.0, [697].log_data[0].max := 1.0, [697].log_data[0].total := 900.0, [697].log_data[0].time := 900.0, [697].log_data[0].minminute := 30, [697].log_data[0].maxminute := 30, [697].log_data[0].valid := 1, [697].log_data[1].valid := 1, [697].log_data[2].valid := 1, [697].log_data[3].valid := 1, [697].log_data[4].valid := 1, [697].log_data[5].valid := 1, [697].log_data[6].valid := 1, [697].log_data[7].valid := 1, [697].log_data[8].valid := 1, [697].log_data[9].valid := 1, [697].log_data[10].valid := 1, [697].log_data[11].valid := 1, [697].log_data[12].valid := 1, [697].log_data[13].valid := 1, [697].log_data[14].valid := 1, [697].log_data[15].valid := 1, [697].log_data[16].valid := 1, [697].log_data[17].valid := 1, [697].log_data[18].valid := 1, [697].log_data[19].valid := 1, [697].time.Year := 2023, [697].time.Month := 1, [697].time.Day := 14, [697].time.Hour := 22, [697].time.Minute := 44, [697].time.Second := 59, [698].log_data[0].min := 1.0, [698].log_data[0].max := 1.0, [698].log_data[0].total := 900.0, [698].log_data[0].time := 900.0, [698].log_data[0].minminute := 45,
        [698].log_data[0].maxminute := 45, [698].log_data[0].valid := 1, [698].log_data[1].valid := 1, [698].log_data[2].valid := 1, [698].log_data[3].valid := 1, [698].log_data[4].valid := 1, [698].log_data[5].valid := 1, [698].log_data[6].valid := 1, [698].log_data[7].valid := 1, [698].log_data[8].valid := 1, [698].log_data[9].valid := 1, [698].log_data[10].valid := 1, [698].log_data[11].valid := 1, [698].log_data[12].valid := 1, [698].log_data[13].valid := 1, [698].log_data[14].valid := 1, [698].log_data[15].valid := 1, [698].log_data[16].valid := 1, [698].log_data[17].valid := 1, [698].log_data[18].valid := 1, [698].log_data[19].valid := 1, [698].time.Year := 2023, [698].time.Month := 1, [698].time.Day := 14, [698].time.Hour := 22, [698].time.Minute := 59, [698].time.Second := 59, [699].log_data[0].min := 1.0, [699].log_data[0].max := 1.0, [699].log_data[0].total := 899.5, [699].log_data[0].time := 899.5, [699].log_data[0].valid := 1, [699].log_data[1].valid := 1, [699].log_data[2].valid := 1, [699].log_data[3].valid := 1, [699].log_data[4].valid := 1, [699].log_data[5].valid := 1, [699].log_data[6].valid := 1, [699].log_data[7].valid := 1, [699].log_data[8].valid := 1, [699].log_data[9].valid := 1, [699].log_data[10].valid := 1, [699].log_data[11].valid := 1, [699].log_data[12].valid := 1, [699].log_data[13].valid := 1, [699].log_data[14].valid := 1, [699].log_data[15].valid := 1, [699].log_data[16].valid := 1, [699].log_data[17].valid := 1, [699].log_data[18].valid := 1, [699].log_data[19].valid := 1, [699].time.Year := 2023, [699].time.Month := 1, [699].time.Day := 14, [699].time.Hour := 23, [699].time.Minute := 14, [699].time.Second := 59, [700].log_data[0].min := 1.0, [700].log_data[0].max := 1.0, [700].log_data[0].total := 900.0,
        [700].log_data[0].time := 900.0, [700].log_data[0].minminute := 15, [700].log_data[0].maxminute := 15, [700].log_data[0].valid := 1, [700].log_data[1].valid := 1, [700].log_data[2].valid := 1, [700].log_data[3].valid := 1, [700].log_data[4].valid := 1, [700].log_data[5].valid := 1, [700].log_data[6].valid := 1, [700].log_data[7].valid := 1, [700].log_data[8].valid := 1, [700].log_data[9].valid := 1, [700].log_data[10].valid := 1, [700].log_data[11].valid := 1, [700].log_data[12].valid := 1, [700].log_data[13].valid := 1, [700].log_data[14].valid := 1, [700].log_data[15].valid := 1, [700].log_data[16].valid := 1, [700].log_data[17].valid := 1, [700].log_data[18].valid := 1, [700].log_data[19].valid := 1, [700].time.Year := 2023, [700].time.Month := 1, [700].time.Day := 14, [700].time.Hour := 23, [700].time.Minute := 29, [700].time.Second := 59, [701].log_data[0].min := 1.0, [701].log_data[0].max := 1.0, [701].log_data[0].total := 900.0, [701].log_data[0].time := 900.0, [701].log_data[0].minminute := 30, [701].log_data[0].maxminute := 30, [701].log_data[0].valid := 1, [701].log_data[1].valid := 1, [701].log_data[2].valid := 1, [701].log_data[3].valid := 1, [701].log_data[4].valid := 1, [701].log_data[5].valid := 1, [701].log_data[6].valid := 1, [701].log_data[7].valid := 1, [701].log_data[8].valid := 1, [701].log_data[9].valid := 1, [701].log_data[10].valid := 1, [701].log_data[11].valid := 1, [701].log_data[12].valid := 1, [701].log_data[13].valid := 1, [701].log_data[14].valid := 1, [701].log_data[15].valid := 1, [701].log_data[16].valid := 1, [701].log_data[17].valid := 1, [701].log_data[18].valid := 1, [701].log_data[19].valid := 1, [701].time.Year := 2023, [701].time.Month := 1, [701].time.Day := 14, [701].time.Hour := 23, [701].time.Minute := 44,
        [701].time.Second := 59, [702].log_data[0].min := 1.0, [702].log_data[0].max := 1.0, [702].log_data[0].total := 900.0, [702].log_data[0].time := 900.0, [702].log_data[0].minminute := 45, [702].log_data[0].maxminute := 45, [702].log_data[0].valid := 1, [702].log_data[1].valid := 1, [702].log_data[2].valid := 1, [702].log_data[3].valid := 1, [702].log_data[4].valid := 1, [702].log_data[5].valid := 1, [702].log_data[6].valid := 1, [702].log_data[7].valid := 1, [702].log_data[8].valid := 1, [702].log_data[9].valid := 1, [702].log_data[10].valid := 1, [702].log_data[11].valid := 1, [702].log_data[12].valid := 1, [702].log_data[13].valid := 1, [702].log_data[14].valid := 1, [702].log_data[15].valid := 1, [702].log_data[16].valid := 1, [702].log_data[17].valid := 1, [702].log_data[18].valid := 1, [702].log_data[19].valid := 1, [702].time.Year := 2023, [702].time.Month := 1, [702].time.Day := 14, [702].time.Hour := 23, [702].time.Minute := 59, [702].time.Second := 59, [703].log_data[0].min := 1.0, [703].log_data[0].max := 1.0, [703].log_data[0].total := 900.0, [703].log_data[0].time := 900.0, [703].log_data[0].valid := 1, [703].log_data[1].valid := 1, [703].log_data[2].valid := 1, [703].log_data[3].valid := 1, [703].log_data[4].valid := 1, [703].log_data[5].valid := 1, [703].log_data[6].valid := 1, [703].log_data[7].valid := 1, [703].log_data[8].valid := 1, [703].log_data[9].valid := 1, [703].log_data[10].valid := 1, [703].log_data[11].valid := 1, [703].log_data[12].valid := 1, [703].log_data[13].valid := 1, [703].log_data[14].valid := 1, [703].log_data[15].valid := 1, [703].log_data[16].valid := 1, [703].log_data[17].valid := 1, [703].log_data[18].valid := 1, [703].log_data[19].valid := 1, [703].time.Year := 2023, [703].time.Month := 1, [703].time.Day := 15,
        [703].time.Minute := 14, [703].time.Second := 59, [704].log_data[0].min := 1.0, [704].log_data[0].max := 1.0, [704].log_data[0].total := 900.0, [704].log_data[0].time := 900.0, [704].log_data[0].minminute := 15, [704].log_data[0].maxminute := 15, [704].log_data[0].valid := 1, [704].log_data[1].valid := 1, [704].log_data[2].valid := 1, [704].log_data[3].valid := 1, [704].log_data[4].valid := 1, [704].log_data[5].valid := 1, [704].log_data[6].valid := 1, [704].log_data[7].valid := 1, [704].log_data[8].valid := 1, [704].log_data[9].valid := 1, [704].log_data[10].valid := 1, [704].log_data[11].valid := 1, [704].log_data[12].valid := 1, [704].log_data[13].valid := 1, [704].log_data[14].valid := 1, [704].log_data[15].valid := 1, [704].log_data[16].valid := 1, [704].log_data[17].valid := 1, [704].log_data[18].valid := 1, [704].log_data[19].valid := 1, [704].time.Year := 2023, [704].time.Month := 1, [704].time.Day := 15, [704].time.Minute := 29, [704].time.Second := 59, [705].log_data[0].min := 1.0, [705].log_data[0].max := 1.0, [705].log_data[0].total := 900.0, [705].log_data[0].time := 900.0, [705].log_data[0].minminute := 30, [705].log_data[0].maxminute := 30, [705].log_data[0].valid := 1, [705].log_data[1].valid := 1, [705].log_data[2].valid := 1, [705].log_data[3].valid := 1, [705].log_data[4].valid := 1, [705].log_data[5].valid := 1, [705].log_data[6].valid := 1, [705].log_data[7].valid := 1, [705].log_data[8].valid := 1, [705].log_data[9].valid := 1, [705].log_data[10].valid := 1, [705].log_data[11].valid := 1, [705].log_data[12].valid := 1, [705].log_data[13].valid := 1, [705].log_data[14].valid := 1, [705].log_data[15].valid := 1, [705].log_data[16].valid := 1, [705].log_data[17].valid := 1, [705].log_data[18].valid := 1, [705].log_data[19].valid := 1, [705].time.Year := 2023,
        [705].time.Month := 1, [705].time.Day := 15, [705].time.Minute := 44, [705].time.Second := 59, [706].log_data[0].min := 1.0, [706].log_data[0].max := 1.0, [706].log_data[0].total := 900.0, [706].log_data[0].time := 900.0, [706].log_data[0].minminute := 45, [706].log_data[0].maxminute := 45, [706].log_data[0].valid := 1, [706].log_data[1].valid := 1, [706].log_data[2].valid := 1, [706].log_data[3].valid := 1, [706].log_data[4].valid := 1, [706].log_data[5].valid := 1, [706].log_data[6].valid := 1, [706].log_data[7].valid := 1, [706].log_data[8].valid := 1, [706].log_data[9].valid := 1, [706].log_data[10].valid := 1, [706].log_data[11].valid := 1, [706].log_data[12].valid := 1, [706].log_data[13].valid := 1, [706].log_data[14].valid := 1, [706].log_data[15].valid := 1, [706].log_data[16].valid := 1, [706].log_data[17].valid := 1, [706].log_data[18].valid := 1, [706].log_data[19].valid := 1, [706].time.Year := 2023, [706].time.Month := 1, [706].time.Day := 15, [706].time.Minute := 59, [706].time.Second := 59, [707].log_data[0].min := 1.0, [707].log_data[0].max := 1.0, [707].log_data[0].total := 900.0, [707].log_data[0].time := 900.0, [707].log_data[0].valid := 1, [707].log_data[1].valid := 1, [707].log_data[2].valid := 1, [707].log_data[3].valid := 1, [707].log_data[4].valid := 1, [707].log_data[5].valid := 1, [707].log_data[6].valid := 1, [707].log_data[7].valid := 1, [707].log_data[8].valid := 1, [707].log_data[9].valid := 1, [707].log_data[10].valid := 1, [707].log_data[11].valid := 1, [707].log_data[12].valid := 1, [707].log_data[13].valid := 1, [707].log_data[14].valid := 1, [707].log_data[15].valid := 1, [707].log_data[16].valid := 1, [707].log_data[17].valid := 1, [707].log_data[18].valid := 1, [707].log_data[19].valid := 1, [707].time.Year := 2023,
        [707].time.Month := 1, [707].time.Day := 15, [707].time.Hour := 1, [707].time.Minute := 14, [707].time.Second := 59, [708].log_data[0].min := 1.0, [708].log_data[0].max := 1.0, [708].log_data[0].total := 900.0, [708].log_data[0].time := 900.0, [708].log_data[0].minminute := 15, [708].log_data[0].maxminute := 15, [708].log_data[0].valid := 1, [708].log_data[1].valid := 1, [708].log_data[2].valid := 1, [708].log_data[3].valid := 1, [708].log_data[4].valid := 1, [708].log_data[5].valid := 1, [708].log_data[6].valid := 1, [708].log_data[7].valid := 1, [708].log_data[8].valid := 1, [708].log_data[9].valid := 1, [708].log_data[10].valid := 1, [708].log_data[11].valid := 1, [708].log_data[12].valid := 1, [708].log_data[13].valid := 1, [708].log_data[14].valid := 1, [708].log_data[15].valid := 1, [708].log_data[16].valid := 1, [708].log_data[17].valid := 1, [708].log_data[18].valid := 1, [708].log_data[19].valid := 1, [708].time.Year := 2023, [708].time.Month := 1, [708].time.Day := 15, [708].time.Hour := 1, [708].time.Minute := 29, [708].time.Second := 59, [709].log_data[0].min := 1.0, [709].log_data[0].max := 1.0, [709].log_data[0].total := 900.0, [709].log_data[0].time := 900.0, [709].log_data[0].minminute := 30, [709].log_data[0].maxminute := 30, [709].log_data[0].valid := 1, [709].log_data[1].valid := 1, [709].log_data[2].valid := 1, [709].log_data[3].valid := 1, [709].log_data[4].valid := 1, [709].log_data[5].valid := 1, [709].log_data[6].valid := 1, [709].log_data[7].valid := 1, [709].log_data[8].valid := 1, [709].log_data[9].valid := 1, [709].log_data[10].valid := 1, [709].log_data[11].valid := 1, [709].log_data[12].valid := 1, [709].log_data[13].valid := 1, [709].log_data[14].valid := 1, [709].log_data[15].valid := 1, [709].log_data[16].valid := 1,
        [709].log_data[17].valid := 1, [709].log_data[18].valid := 1, [709].log_data[19].valid := 1, [709].time.Year := 2023, [709].time.Month := 1, [709].time.Day := 15, [709].time.Hour := 1, [709].time.Minute := 44, [709].time.Second := 59, [710].log_data[0].min := 1.0, [710].log_data[0].max := 1.0, [710].log_data[0].total := 900.0, [710].log_data[0].time := 900.0, [710].log_data[0].minminute := 45, [710].log_data[0].maxminute := 45, [710].log_data[0].valid := 1, [710].log_data[1].valid := 1, [710].log_data[2].valid := 1, [710].log_data[3].valid := 1, [710].log_data[4].valid := 1, [710].log_data[5].valid := 1, [710].log_data[6].valid := 1, [710].log_data[7].valid := 1, [710].log_data[8].valid := 1, [710].log_data[9].valid := 1, [710].log_data[10].valid := 1, [710].log_data[11].valid := 1, [710].log_data[12].valid := 1, [710].log_data[13].valid := 1, [710].log_data[14].valid := 1, [710].log_data[15].valid := 1, [710].log_data[16].valid := 1, [710].log_data[17].valid := 1, [710].log_data[18].valid := 1, [710].log_data[19].valid := 1, [710].time.Year := 2023, [710].time.Month := 1, [710].time.Day := 15, [710].time.Hour := 1, [710].time.Minute := 59, [710].time.Second := 59, [711].log_data[0].min := 1.0, [711].log_data[0].max := 1.0, [711].log_data[0].total := 900.0, [711].log_data[0].time := 900.0, [711].log_data[0].valid := 1, [711].log_data[1].valid := 1, [711].log_data[2].valid := 1, [711].log_data[3].valid := 1, [711].log_data[4].valid := 1, [711].log_data[5].valid := 1, [711].log_data[6].valid := 1, [711].log_data[7].valid := 1, [711].log_data[8].valid := 1, [711].log_data[9].valid := 1, [711].log_data[10].valid := 1, [711].log_data[11].valid := 1, [711].log_data[12].valid := 1, [711].log_data[13].valid := 1, [711].log_data[14].valid := 1,
        [711].log_data[15].valid := 1, [711].log_data[16].valid := 1, [711].log_data[17].valid := 1, [711].log_data[18].valid := 1, [711].log_data[19].valid := 1, [711].time.Year := 2023, [711].time.Month := 1, [711].time.Day := 15, [711].time.Hour := 2, [711].time.Minute := 14, [711].time.Second := 59, [712].log_data[0].min := 1.0, [712].log_data[0].max := 1.0, [712].log_data[0].total := 900.0, [712].log_data[0].time := 900.0, [712].log_data[0].minminute := 15, [712].log_data[0].maxminute := 15, [712].log_data[0].valid := 1, [712].log_data[1].valid := 1, [712].log_data[2].valid := 1, [712].log_data[3].valid := 1, [712].log_data[4].valid := 1, [712].log_data[5].valid := 1, [712].log_data[6].valid := 1, [712].log_data[7].valid := 1, [712].log_data[8].valid := 1, [712].log_data[9].valid := 1, [712].log_data[10].valid := 1, [712].log_data[11].valid := 1, [712].log_data[12].valid := 1, [712].log_data[13].valid := 1, [712].log_data[14].valid := 1, [712].log_data[15].valid := 1, [712].log_data[16].valid := 1, [712].log_data[17].valid := 1, [712].log_data[18].valid := 1, [712].log_data[19].valid := 1, [712].time.Year := 2023, [712].time.Month := 1, [712].time.Day := 15, [712].time.Hour := 2, [712].time.Minute := 29, [712].time.Second := 59, [713].log_data[0].min := 1.0, [713].log_data[0].max := 1.0, [713].log_data[0].total := 900.0, [713].log_data[0].time := 900.0, [713].log_data[0].minminute := 30, [713].log_data[0].maxminute := 30, [713].log_data[0].valid := 1, [713].log_data[1].valid := 1, [713].log_data[2].valid := 1, [713].log_data[3].valid := 1, [713].log_data[4].valid := 1, [713].log_data[5].valid := 1, [713].log_data[6].valid := 1, [713].log_data[7].valid := 1, [713].log_data[8].valid := 1, [713].log_data[9].valid := 1, [713].log_data[10].valid := 1,
        [713].log_data[11].valid := 1, [713].log_data[12].valid := 1, [713].log_data[13].valid := 1, [713].log_data[14].valid := 1, [713].log_data[15].valid := 1, [713].log_data[16].valid := 1, [713].log_data[17].valid := 1, [713].log_data[18].valid := 1, [713].log_data[19].valid := 1, [713].time.Year := 2023, [713].time.Month := 1, [713].time.Day := 15, [713].time.Hour := 2, [713].time.Minute := 44, [713].time.Second := 59, [714].log_data[0].min := 1.0, [714].log_data[0].max := 1.0, [714].log_data[0].total := 900.0, [714].log_data[0].time := 900.0, [714].log_data[0].minminute := 45, [714].log_data[0].maxminute := 45, [714].log_data[0].valid := 1, [714].log_data[1].valid := 1, [714].log_data[2].valid := 1, [714].log_data[3].valid := 1, [714].log_data[4].valid := 1, [714].log_data[5].valid := 1, [714].log_data[6].valid := 1, [714].log_data[7].valid := 1, [714].log_data[8].valid := 1, [714].log_data[9].valid := 1, [714].log_data[10].valid := 1, [714].log_data[11].valid := 1, [714].log_data[12].valid := 1, [714].log_data[13].valid := 1, [714].log_data[14].valid := 1, [714].log_data[15].valid := 1, [714].log_data[16].valid := 1, [714].log_data[17].valid := 1, [714].log_data[18].valid := 1, [714].log_data[19].valid := 1, [714].time.Year := 2023, [714].time.Month := 1, [714].time.Day := 15, [714].time.Hour := 2, [714].time.Minute := 59, [714].time.Second := 59, [715].log_data[0].min := 1.0, [715].log_data[0].max := 1.0, [715].log_data[0].total := 900.0, [715].log_data[0].time := 900.0, [715].log_data[0].valid := 1, [715].log_data[1].valid := 1, [715].log_data[2].valid := 1, [715].log_data[3].valid := 1, [715].log_data[4].valid := 1, [715].log_data[5].valid := 1, [715].log_data[6].valid := 1, [715].log_data[7].valid := 1, [715].log_data[8].valid := 1,
        [715].log_data[9].valid := 1, [715].log_data[10].valid := 1, [715].log_data[11].valid := 1, [715].log_data[12].valid := 1, [715].log_data[13].valid := 1, [715].log_data[14].valid := 1, [715].log_data[15].valid := 1, [715].log_data[16].valid := 1, [715].log_data[17].valid := 1, [715].log_data[18].valid := 1, [715].log_data[19].valid := 1, [715].time.Year := 2023, [715].time.Month := 1, [715].time.Day := 15, [715].time.Hour := 3, [715].time.Minute := 14, [715].time.Second := 59, [716].log_data[0].min := 1.0, [716].log_data[0].max := 1.0, [716].log_data[0].total := 900.0, [716].log_data[0].time := 900.0, [716].log_data[0].minminute := 15, [716].log_data[0].maxminute := 15, [716].log_data[0].valid := 1, [716].log_data[1].valid := 1, [716].log_data[2].valid := 1, [716].log_data[3].valid := 1, [716].log_data[4].valid := 1, [716].log_data[5].valid := 1, [716].log_data[6].valid := 1, [716].log_data[7].valid := 1, [716].log_data[8].valid := 1, [716].log_data[9].valid := 1, [716].log_data[10].valid := 1, [716].log_data[11].valid := 1, [716].log_data[12].valid := 1, [716].log_data[13].valid := 1, [716].log_data[14].valid := 1, [716].log_data[15].valid := 1, [716].log_data[16].valid := 1, [716].log_data[17].valid := 1, [716].log_data[18].valid := 1, [716].log_data[19].valid := 1, [716].time.Year := 2023, [716].time.Month := 1, [716].time.Day := 15, [716].time.Hour := 3, [716].time.Minute := 29, [716].time.Second := 59, [717].log_data[0].min := 1.0, [717].log_data[0].max := 1.0, [717].log_data[0].total := 900.0, [717].log_data[0].time := 900.0, [717].log_data[0].minminute := 30, [717].log_data[0].maxminute := 30, [717].log_data[0].valid := 1, [717].log_data[1].valid := 1, [717].log_data[2].valid := 1, [717].log_data[3].valid := 1, [717].log_data[4].valid := 1,
        [717].log_data[5].valid := 1, [717].log_data[6].valid := 1, [717].log_data[7].valid := 1, [717].log_data[8].valid := 1, [717].log_data[9].valid := 1, [717].log_data[10].valid := 1, [717].log_data[11].valid := 1, [717].log_data[12].valid := 1, [717].log_data[13].valid := 1, [717].log_data[14].valid := 1, [717].log_data[15].valid := 1, [717].log_data[16].valid := 1, [717].log_data[17].valid := 1, [717].log_data[18].valid := 1, [717].log_data[19].valid := 1, [717].time.Year := 2023, [717].time.Month := 1, [717].time.Day := 15, [717].time.Hour := 3, [717].time.Minute := 44, [717].time.Second := 59, [718].log_data[0].min := 1.0, [718].log_data[0].max := 1.0, [718].log_data[0].total := 900.0, [718].log_data[0].time := 900.0, [718].log_data[0].minminute := 45, [718].log_data[0].maxminute := 45, [718].log_data[0].valid := 1, [718].log_data[1].valid := 1, [718].log_data[2].valid := 1, [718].log_data[3].valid := 1, [718].log_data[4].valid := 1, [718].log_data[5].valid := 1, [718].log_data[6].valid := 1, [718].log_data[7].valid := 1, [718].log_data[8].valid := 1, [718].log_data[9].valid := 1, [718].log_data[10].valid := 1, [718].log_data[11].valid := 1, [718].log_data[12].valid := 1, [718].log_data[13].valid := 1, [718].log_data[14].valid := 1, [718].log_data[15].valid := 1, [718].log_data[16].valid := 1, [718].log_data[17].valid := 1, [718].log_data[18].valid := 1, [718].log_data[19].valid := 1, [718].time.Year := 2023, [718].time.Month := 1, [718].time.Day := 15, [718].time.Hour := 3, [718].time.Minute := 59, [718].time.Second := 59, [719].log_data[0].min := 1.0, [719].log_data[0].max := 1.0, [719].log_data[0].total := 900.0, [719].log_data[0].time := 900.0, [719].log_data[0].valid := 1, [719].log_data[1].valid := 1, [719].log_data[2].valid := 1,
        [719].log_data[3].valid := 1, [719].log_data[4].valid := 1, [719].log_data[5].valid := 1, [719].log_data[6].valid := 1, [719].log_data[7].valid := 1, [719].log_data[8].valid := 1, [719].log_data[9].valid := 1, [719].log_data[10].valid := 1, [719].log_data[11].valid := 1, [719].log_data[12].valid := 1, [719].log_data[13].valid := 1, [719].log_data[14].valid := 1, [719].log_data[15].valid := 1, [719].log_data[16].valid := 1, [719].log_data[17].valid := 1, [719].log_data[18].valid := 1, [719].log_data[19].valid := 1, [719].time.Year := 2023, [719].time.Month := 1, [719].time.Day := 15, [719].time.Hour := 4, [719].time.Minute := 14, [719].time.Second := 59, [720].log_data[0].min := 1.0, [720].log_data[0].max := 1.0, [720].log_data[0].total := 900.0, [720].log_data[0].time := 900.0, [720].log_data[0].minminute := 15, [720].log_data[0].maxminute := 15, [720].log_data[0].valid := 1, [720].log_data[1].valid := 1, [720].log_data[2].valid := 1, [720].log_data[3].valid := 1, [720].log_data[4].valid := 1, [720].log_data[5].valid := 1, [720].log_data[6].valid := 1, [720].log_data[7].valid := 1, [720].log_data[8].valid := 1, [720].log_data[9].valid := 1, [720].log_data[10].valid := 1, [720].log_data[11].valid := 1, [720].log_data[12].valid := 1, [720].log_data[13].valid := 1, [720].log_data[14].valid := 1, [720].log_data[15].valid := 1, [720].log_data[16].valid := 1, [720].log_data[17].valid := 1, [720].log_data[18].valid := 1, [720].log_data[19].valid := 1, [720].time.Year := 2023, [720].time.Month := 1, [720].time.Day := 15, [720].time.Hour := 4, [720].time.Minute := 29, [720].time.Second := 59, [721].log_data[0].min := 1.0, [721].log_data[0].max := 1.0, [721].log_data[0].total := 900.0, [721].log_data[0].time := 900.0, [721].log_data[0].minminute := 30,
        [721].log_data[0].maxminute := 30, [721].log_data[0].valid := 1, [721].log_data[1].valid := 1, [721].log_data[2].valid := 1, [721].log_data[3].valid := 1, [721].log_data[4].valid := 1, [721].log_data[5].valid := 1, [721].log_data[6].valid := 1, [721].log_data[7].valid := 1, [721].log_data[8].valid := 1, [721].log_data[9].valid := 1, [721].log_data[10].valid := 1, [721].log_data[11].valid := 1, [721].log_data[12].valid := 1, [721].log_data[13].valid := 1, [721].log_data[14].valid := 1, [721].log_data[15].valid := 1, [721].log_data[16].valid := 1, [721].log_data[17].valid := 1, [721].log_data[18].valid := 1, [721].log_data[19].valid := 1, [721].time.Year := 2023, [721].time.Month := 1, [721].time.Day := 15, [721].time.Hour := 4, [721].time.Minute := 44, [721].time.Second := 59, [722].log_data[0].min := 1.0, [722].log_data[0].max := 1.0, [722].log_data[0].total := 900.0, [722].log_data[0].time := 900.0, [722].log_data[0].minminute := 45, [722].log_data[0].maxminute := 45, [722].log_data[0].valid := 1, [722].log_data[1].valid := 1, [722].log_data[2].valid := 1, [722].log_data[3].valid := 1, [722].log_data[4].valid := 1, [722].log_data[5].valid := 1, [722].log_data[6].valid := 1, [722].log_data[7].valid := 1, [722].log_data[8].valid := 1, [722].log_data[9].valid := 1, [722].log_data[10].valid := 1, [722].log_data[11].valid := 1, [722].log_data[12].valid := 1, [722].log_data[13].valid := 1, [722].log_data[14].valid := 1, [722].log_data[15].valid := 1, [722].log_data[16].valid := 1, [722].log_data[17].valid := 1, [722].log_data[18].valid := 1, [722].log_data[19].valid := 1, [722].time.Year := 2023, [722].time.Month := 1, [722].time.Day := 15, [722].time.Hour := 4, [722].time.Minute := 59, [722].time.Second := 59, [723].log_data[0].min := 1.0,
        [723].log_data[0].max := 1.0, [723].log_data[0].total := 900.0, [723].log_data[0].time := 900.0, [723].log_data[0].valid := 1, [723].log_data[1].valid := 1, [723].log_data[2].valid := 1, [723].log_data[3].valid := 1, [723].log_data[4].valid := 1, [723].log_data[5].valid := 1, [723].log_data[6].valid := 1, [723].log_data[7].valid := 1, [723].log_data[8].valid := 1, [723].log_data[9].valid := 1, [723].log_data[10].valid := 1, [723].log_data[11].valid := 1, [723].log_data[12].valid := 1, [723].log_data[13].valid := 1, [723].log_data[14].valid := 1, [723].log_data[15].valid := 1, [723].log_data[16].valid := 1, [723].log_data[17].valid := 1, [723].log_data[18].valid := 1, [723].log_data[19].valid := 1, [723].time.Year := 2023, [723].time.Month := 1, [723].time.Day := 15, [723].time.Hour := 5, [723].time.Minute := 14, [723].time.Second := 59, [724].log_data[0].min := 1.0, [724].log_data[0].max := 1.0, [724].log_data[0].total := 900.0, [724].log_data[0].time := 900.0, [724].log_data[0].minminute := 15, [724].log_data[0].maxminute := 15, [724].log_data[0].valid := 1, [724].log_data[1].valid := 1, [724].log_data[2].valid := 1, [724].log_data[3].valid := 1, [724].log_data[4].valid := 1, [724].log_data[5].valid := 1, [724].log_data[6].valid := 1, [724].log_data[7].valid := 1, [724].log_data[8].valid := 1, [724].log_data[9].valid := 1, [724].log_data[10].valid := 1, [724].log_data[11].valid := 1, [724].log_data[12].valid := 1, [724].log_data[13].valid := 1, [724].log_data[14].valid := 1, [724].log_data[15].valid := 1, [724].log_data[16].valid := 1, [724].log_data[17].valid := 1, [724].log_data[18].valid := 1, [724].log_data[19].valid := 1, [724].time.Year := 2023, [724].time.Month := 1, [724].time.Day := 15, [724].time.Hour := 5, [724].time.Minute := 29,
        [724].time.Second := 59, [725].log_data[0].min := 1.0, [725].log_data[0].max := 1.0, [725].log_data[0].total := 900.0, [725].log_data[0].time := 900.0, [725].log_data[0].minminute := 30, [725].log_data[0].maxminute := 30, [725].log_data[0].valid := 1, [725].log_data[1].valid := 1, [725].log_data[2].valid := 1, [725].log_data[3].valid := 1, [725].log_data[4].valid := 1, [725].log_data[5].valid := 1, [725].log_data[6].valid := 1, [725].log_data[7].valid := 1, [725].log_data[8].valid := 1, [725].log_data[9].valid := 1, [725].log_data[10].valid := 1, [725].log_data[11].valid := 1, [725].log_data[12].valid := 1, [725].log_data[13].valid := 1, [725].log_data[14].valid := 1, [725].log_data[15].valid := 1, [725].log_data[16].valid := 1, [725].log_data[17].valid := 1, [725].log_data[18].valid := 1, [725].log_data[19].valid := 1, [725].time.Year := 2023, [725].time.Month := 1, [725].time.Day := 15, [725].time.Hour := 5, [725].time.Minute := 44, [725].time.Second := 59, [726].log_data[0].min := 1.0, [726].log_data[0].max := 1.0, [726].log_data[0].total := 900.0, [726].log_data[0].time := 900.0, [726].log_data[0].minminute := 45, [726].log_data[0].maxminute := 45, [726].log_data[0].valid := 1, [726].log_data[1].valid := 1, [726].log_data[2].valid := 1, [726].log_data[3].valid := 1, [726].log_data[4].valid := 1, [726].log_data[5].valid := 1, [726].log_data[6].valid := 1, [726].log_data[7].valid := 1, [726].log_data[8].valid := 1, [726].log_data[9].valid := 1, [726].log_data[10].valid := 1, [726].log_data[11].valid := 1, [726].log_data[12].valid := 1, [726].log_data[13].valid := 1, [726].log_data[14].valid := 1, [726].log_data[15].valid := 1, [726].log_data[16].valid := 1, [726].log_data[17].valid := 1, [726].log_data[18].valid := 1, [726].log_data[19].valid := 1, [726].time.Year := 2023,
        [726].time.Month := 1, [726].time.Day := 15, [726].time.Hour := 5, [726].time.Minute := 59, [726].time.Second := 59, [727].log_data[0].min := 1.0, [727].log_data[0].max := 1.0, [727].log_data[0].total := 900.0, [727].log_data[0].time := 900.0, [727].log_data[0].valid := 1, [727].log_data[1].valid := 1, [727].log_data[2].valid := 1, [727].log_data[3].valid := 1, [727].log_data[4].valid := 1, [727].log_data[5].valid := 1, [727].log_data[6].valid := 1, [727].log_data[7].valid := 1, [727].log_data[8].valid := 1, [727].log_data[9].valid := 1, [727].log_data[10].valid := 1, [727].log_data[11].valid := 1, [727].log_data[12].valid := 1, [727].log_data[13].valid := 1, [727].log_data[14].valid := 1, [727].log_data[15].valid := 1, [727].log_data[16].valid := 1, [727].log_data[17].valid := 1, [727].log_data[18].valid := 1, [727].log_data[19].valid := 1, [727].time.Year := 2023, [727].time.Month := 1, [727].time.Day := 15, [727].time.Hour := 6, [727].time.Minute := 14, [727].time.Second := 59, [728].log_data[0].min := 1.0, [728].log_data[0].max := 1.0, [728].log_data[0].total := 900.0, [728].log_data[0].time := 900.0, [728].log_data[0].minminute := 15, [728].log_data[0].maxminute := 15, [728].log_data[0].valid := 1, [728].log_data[1].valid := 1, [728].log_data[2].valid := 1, [728].log_data[3].valid := 1, [728].log_data[4].valid := 1, [728].log_data[5].valid := 1, [728].log_data[6].valid := 1, [728].log_data[7].valid := 1, [728].log_data[8].valid := 1, [728].log_data[9].valid := 1, [728].log_data[10].valid := 1, [728].log_data[11].valid := 1, [728].log_data[12].valid := 1, [728].log_data[13].valid := 1, [728].log_data[14].valid := 1, [728].log_data[15].valid := 1, [728].log_data[16].valid := 1, [728].log_data[17].valid := 1, [728].log_data[18].valid := 1,
        [728].log_data[19].valid := 1, [728].time.Year := 2023, [728].time.Month := 1, [728].time.Day := 15, [728].time.Hour := 6, [728].time.Minute := 29, [728].time.Second := 59, [729].log_data[0].min := 1.0, [729].log_data[0].max := 1.0, [729].log_data[0].total := 900.0, [729].log_data[0].time := 900.0, [729].log_data[0].minminute := 30, [729].log_data[0].maxminute := 30, [729].log_data[0].valid := 1, [729].log_data[1].valid := 1, [729].log_data[2].valid := 1, [729].log_data[3].valid := 1, [729].log_data[4].valid := 1, [729].log_data[5].valid := 1, [729].log_data[6].valid := 1, [729].log_data[7].valid := 1, [729].log_data[8].valid := 1, [729].log_data[9].valid := 1, [729].log_data[10].valid := 1, [729].log_data[11].valid := 1, [729].log_data[12].valid := 1, [729].log_data[13].valid := 1, [729].log_data[14].valid := 1, [729].log_data[15].valid := 1, [729].log_data[16].valid := 1, [729].log_data[17].valid := 1, [729].log_data[18].valid := 1, [729].log_data[19].valid := 1, [729].time.Year := 2023, [729].time.Month := 1, [729].time.Day := 15, [729].time.Hour := 6, [729].time.Minute := 44, [729].time.Second := 59, [730].log_data[0].min := 1.0, [730].log_data[0].max := 1.0, [730].log_data[0].total := 900.0, [730].log_data[0].time := 900.0, [730].log_data[0].minminute := 45, [730].log_data[0].maxminute := 45, [730].log_data[0].valid := 1, [730].log_data[1].valid := 1, [730].log_data[2].valid := 1, [730].log_data[3].valid := 1, [730].log_data[4].valid := 1, [730].log_data[5].valid := 1, [730].log_data[6].valid := 1, [730].log_data[7].valid := 1, [730].log_data[8].valid := 1, [730].log_data[9].valid := 1, [730].log_data[10].valid := 1, [730].log_data[11].valid := 1, [730].log_data[12].valid := 1, [730].log_data[13].valid := 1, [730].log_data[14].valid := 1,
        [730].log_data[15].valid := 1, [730].log_data[16].valid := 1, [730].log_data[17].valid := 1, [730].log_data[18].valid := 1, [730].log_data[19].valid := 1, [730].time.Year := 2023, [730].time.Month := 1, [730].time.Day := 15, [730].time.Hour := 6, [730].time.Minute := 59, [730].time.Second := 59, [731].log_data[0].min := 1.0, [731].log_data[0].max := 1.0, [731].log_data[0].total := 900.0, [731].log_data[0].time := 900.0, [731].log_data[0].valid := 1, [731].log_data[1].valid := 1, [731].log_data[2].valid := 1, [731].log_data[3].valid := 1, [731].log_data[4].valid := 1, [731].log_data[5].valid := 1, [731].log_data[6].valid := 1, [731].log_data[7].valid := 1, [731].log_data[8].valid := 1, [731].log_data[9].valid := 1, [731].log_data[10].valid := 1, [731].log_data[11].valid := 1, [731].log_data[12].valid := 1, [731].log_data[13].valid := 1, [731].log_data[14].valid := 1, [731].log_data[15].valid := 1, [731].log_data[16].valid := 1, [731].log_data[17].valid := 1, [731].log_data[18].valid := 1, [731].log_data[19].valid := 1, [731].time.Year := 2023, [731].time.Month := 1, [731].time.Day := 15, [731].time.Hour := 7, [731].time.Minute := 14, [731].time.Second := 59, [732].log_data[0].min := 1.0, [732].log_data[0].max := 1.0, [732].log_data[0].total := 900.0, [732].log_data[0].time := 900.0, [732].log_data[0].minminute := 15, [732].log_data[0].maxminute := 15, [732].log_data[0].valid := 1, [732].log_data[1].valid := 1, [732].log_data[2].valid := 1, [732].log_data[3].valid := 1, [732].log_data[4].valid := 1, [732].log_data[5].valid := 1, [732].log_data[6].valid := 1, [732].log_data[7].valid := 1, [732].log_data[8].valid := 1, [732].log_data[9].valid := 1, [732].log_data[10].valid := 1, [732].log_data[11].valid := 1, [732].log_data[12].valid := 1,
        [732].log_data[13].valid := 1, [732].log_data[14].valid := 1, [732].log_data[15].valid := 1, [732].log_data[16].valid := 1, [732].log_data[17].valid := 1, [732].log_data[18].valid := 1, [732].log_data[19].valid := 1, [732].time.Year := 2023, [732].time.Month := 1, [732].time.Day := 15, [732].time.Hour := 7, [732].time.Minute := 29, [732].time.Second := 59, [733].log_data[0].min := 1.0, [733].log_data[0].max := 1.0, [733].log_data[0].total := 900.0, [733].log_data[0].time := 900.0, [733].log_data[0].minminute := 30, [733].log_data[0].maxminute := 30, [733].log_data[0].valid := 1, [733].log_data[1].valid := 1, [733].log_data[2].valid := 1, [733].log_data[3].valid := 1, [733].log_data[4].valid := 1, [733].log_data[5].valid := 1, [733].log_data[6].valid := 1, [733].log_data[7].valid := 1, [733].log_data[8].valid := 1, [733].log_data[9].valid := 1, [733].log_data[10].valid := 1, [733].log_data[11].valid := 1, [733].log_data[12].valid := 1, [733].log_data[13].valid := 1, [733].log_data[14].valid := 1, [733].log_data[15].valid := 1, [733].log_data[16].valid := 1, [733].log_data[17].valid := 1, [733].log_data[18].valid := 1, [733].log_data[19].valid := 1, [733].time.Year := 2023, [733].time.Month := 1, [733].time.Day := 15, [733].time.Hour := 7, [733].time.Minute := 44, [733].time.Second := 59, [734].log_data[0].min := 1.0, [734].log_data[0].max := 1.0, [734].log_data[0].total := 900.0, [734].log_data[0].time := 900.0, [734].log_data[0].minminute := 45, [734].log_data[0].maxminute := 45, [734].log_data[0].valid := 1, [734].log_data[1].valid := 1, [734].log_data[2].valid := 1, [734].log_data[3].valid := 1, [734].log_data[4].valid := 1, [734].log_data[5].valid := 1, [734].log_data[6].valid := 1, [734].log_data[7].valid := 1, [734].log_data[8].valid := 1,
